# B&R Automation Studio project RTFProj
Automation Studio 4.2.10.53 SP; technology packages: mapp 1.60.1, mappView 1.3.1, TextSystem 

## Configuration RTFProjRG

CPU 5PPC2100.BY44-000, AutomationRuntime B4.26, Build 4.1.2, Vc not used, Safety 1.10

### Task classes (Cpu.sw)
```
Cyclic#1 (cycle 2000 us, tolerance 0 us):
  table_foot <- Real_Game.Technology.table_football.prg
Cyclic#4 (cycle 100000 us, tolerance 100000 us):
  Client <- Connection.Client.prg
DataObjects: assl1, Arnc0sys, Acp10sys
NcDataObjects: acp10etxen <- ACP10_ETXEN.acp10etxen.dob, rotaryFWa <- Real_Game.Motion.rotaryFWobj.rotaryFWa.dob, rotaryFWi <- Real_Game.Motion.rotaryFWobj.rotaryFWi.dob, rotaryMDa <- Real_Game.Motion.rotaryMDobj.rotaryMDa.dob, rotaryMDi <- Real_Game.Motion.rotaryMDobj.rotaryMDi.dob, linearFWa <- Real_Game.Motion.linearFWobj.linearFWa.dob, linearFWi <- Real_Game.Motion.linearFWobj.linearFWi.dob, linearMDa <- Real_Game.Motion.linearMDobj.linearMDa.dob, linearMDi <- Real_Game.Motion.linearMDobj.linearMDi.dob, rotDFa <- Real_Game.Motion.rotDFobj.rotDFa.dob, rotDFi <- Real_Game.Motion.rotDFobj.rotDFi.dob, rotDFVa <- Real_Game.Motion.rotDFVobj.rotDFVa.dob, rotDFVi <- Real_Game.Motion.rotDFVobj.rotDFVi.dob, rotGKa <- Real_Game.Motion.rotGKobj.rotGKa.dob, rotGKi <- Real_Game.Motion.rotGKobj.rotGKi.dob, linDFa <- Real_Game.Motion.linDFobj.linDFa.dob, linDFi <- Real_Game.Motion.linDFobj.linDFi.dob, linDFVa <- Real_Game.Motion.linDFVobj.linDFVa.dob, linDFVi <- Real_Game.Motion.linDFVobj.linDFVi.dob, linGKa <- Real_Game.Motion.linGKobj.linGKa.dob, linGKi <- Real_Game.Motion.linGKobj.linGKi.dob
Binaries: arsvcreg, mvLoader, TCData, udbdef, Linear, iomap, OpcUaMap, sysconf, Config, TC, Config_1, ashwd, asfw, User, arconfig, Role, Rotary, Acp10map, acp10cfg, Arnc0map, arnc0cfg
Libraries: operator, runtime, AsIecCon, sys_lib, astime, AsArSdm, AsWStr, asstring, DataObj, AsArLog, FileIO, AsArProf, AsMem, brsystem, standard, rp_funcx1, GoalKeeper, AsBrStr, IecCheck, MTTypes, MpCom, MpAlarmX, MTBasics, AsSafety, AsXml, MpAxis, Acp10_MC, Acp10man, NcGlobal, Acp10par, RO_Sensors, Camera, Bar_Light, AsUDP, powerlnk, areventlog
```

### Hardware
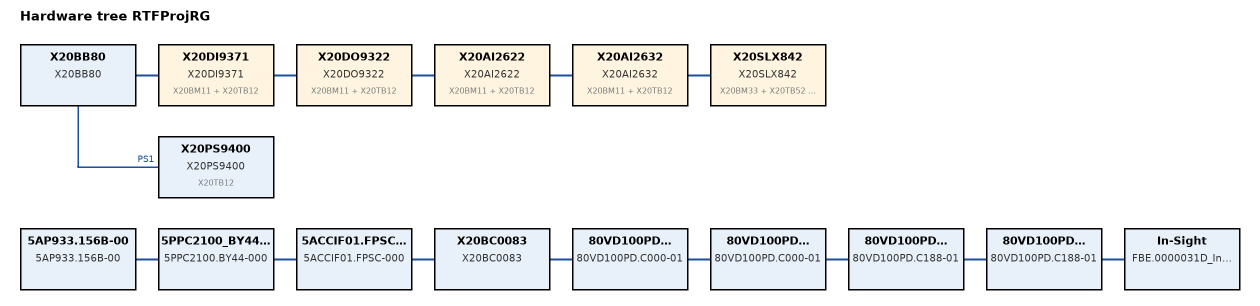
```
5ACCIF01.FPSC-000 : 5ACCIF01.FPSC-000 v1.2.1.0  [SL -> 5PPC2100_BY44_000.SL1]
  Connector IF1:
    Channel1
    ChannelID1 = ACP10_MC_BROADCAST
    ChannelType1 = OCTET[96]
5AP933.156B-00 : 5AP933.156B-00 v1.4.0.1
5PPC2100_BY44_000 : 5PPC2100.BY44-000 v1.2.4.0  [SY -> 5AP933.156B-00.SY1]
  Connector IF3:
    ActivateDevice = 1
  AutomationRuntime = AR010
  ConfigurationID = RTFProj_Config1
  TimerDeviceType = EPLX2X
  TimerDevice = 5ACCIF01.FPSC-000.IF1
  TaskClassIdleTime = 2000
  Cyclic1Duration = 2000
  Cyclic1Tolerance = 0
  Cyclic2Duration = 10000
  Cyclic2Tolerance = 10000
  Cyclic3Duration = 50000
  Cyclic3Tolerance = 50000
  Cyclic4Duration = 100000
  Cyclic4Tolerance = 100000
  Cyclic5Duration = 200000
  Cyclic5Tolerance = 200000
  Cyclic6Duration = 500000
  Cyclic6Tolerance = 500000
  Cyclic7Duration = 1000000
  Cyclic7Tolerance = 1000000
  Cyclic8Duration = 10000
  Cyclic8Tolerance = 30000000
  ActivateOpcUa = 1
  OpcUa_Security_SoftwareCertificates = 
80VD100PD.C000-01 : 80VD100PD.C000-01 v2.0.1.0  [PLK1 -> X20BC0083.PLK2 (NodeNumber=2); PLK2 -> 80VD100PD.C000-01a.PLK1 (NodeNumber=2)]
  BothEndSwitchesAreNormallyOpen_r1 = on
  QuickStopIsNormallyOpen_r1 = on
  BothEndSwitchesAreNormallyOpen_r2 = on
  QuickStopIsNormallyOpen_r2 = on
80VD100PD.C000-01a : 80VD100PD.C000-01 v2.0.1.0  [PLK1 -> 80VD100PD.C000-01.PLK2 (NodeNumber=4); PLK2 -> 80VD100PD.C188-01.PLK1 (NodeNumber=4)]
  BothEndSwitchesAreNormallyOpen_r1 = on
  QuickStopIsNormallyOpen_r1 = on
  BothEndSwitchesAreNormallyOpen_r2 = on
  QuickStopIsNormallyOpen_r2 = on
80VD100PD.C188-01 : 80VD100PD.C188-01 v2.0.1.0  [PLK1 -> 80VD100PD.C000-01a.PLK2 (NodeNumber=3); PLK2 -> 80VD100PD.C188-01a.PLK1 (NodeNumber=3)]
  BothEndSwitchesAreNormallyOpen_r1 = on
  QuickStopIsNormallyOpen_r1 = on
  BothEndSwitchesAreNormallyOpen_r2 = on
  QuickStopIsNormallyOpen_r2 = on
80VD100PD.C188-01a : 80VD100PD.C188-01 v2.0.1.0  [PLK1 -> 80VD100PD.C188-01.PLK2 (NodeNumber=5); PLK2 -> In-Sight.PLK1 (NodeNumber=5)]
  BothEndSwitchesAreNormallyOpen_r1 = on
  QuickStopIsNormallyOpen_r1 = on
  BothEndSwitchesAreNormallyOpen_r2 = on
  QuickStopIsNormallyOpen_r2 = on
In-Sight : FBE.0000031D_In-Sight-7000 v4.8.0 (OrderNumber=In-Sight)  [PLK1 -> 80VD100PD.C188-01a.PLK2 (NodeNumber=6)]
  Supervision = off
  p2000s01_direction = wo
  p2000s02_direction = wo
  p2001s01_direction = ro
  p2001s02_direction = ro
  p2001s03_direction = ro
  p2010s02_direction = ro
  p2011s01_direction = ro
  p2011s02_direction = ro
  p2011s03_direction = ro
  p2011s04_direction = ro
  p2021s01_direction = wo
X20AI2622 : X20AI2622 v1.0.3.1  [SS1 -> X20TB12c.SS; SL -> X20BM11b.SL1]
  Supervision = off
  ChannelType01 = 4 to 20mA
  ChannelType02 = 4 to 20mA
X20AI2632 : X20AI2632 v1.1.5.1  [SS1 -> X20TB12d.SS; SL -> X20BM11c.SL1]
  ChannelType01 = 0 to 20mA
  ChannelType02 = 0 to 20mA
X20BB80 : X20BB80 v1.0.0.2
X20BC0083 : X20BC0083 v2.5.2.0  [PLK1 -> 5ACCIF01.FPSC-000.IF1 (NodeNumber=1); PLK2 -> 80VD100PD.C000-01.PLK1 (NodeNumber=1); SL -> X20BB80.SL1]
  Supervision = off
X20BM11 : X20BM11 v1.0.0.1  [X2X1 -> X20BB80.IF1]
X20BM11a : X20BM11 v1.0.0.1  [X2X1 -> X20BM11.X2X2]
X20BM11b : X20BM11 v1.0.0.1  [X2X1 -> X20BM11a.X2X2]
X20BM11c : X20BM11 v1.0.0.1  [X2X1 -> X20BM11b.X2X2]
X20BM33 : X20BM33 v1.0.0.4  [X2X1 -> X20BM11c.X2X2]
X20DI9371 : X20DI9371 v1.0.1.3  [SS1 -> X20TB12a.SS; SL -> X20BM11.SL1]
  Supervision = off
X20DO9322 : X20DO9322 v1.0.3.0  [SS1 -> X20TB12b.SS; SL -> X20BM11a.SL1]
  Supervision = off
X20PS9400 : X20PS9400 v1.0.2.4  [SS1 -> X20TB12.SS; PS -> X20BB80.PS1]
  Supervision = off
X20SLX842 : X20SLX842 v1.10.3.1  [SS1 -> X20TB52.SS; SS2 -> X20TB52a.SS; SL -> X20BM33.SL1]
  SafeProject = SafeLOGIC-1
  SafeDesigner = 4.2.2.18
  DigitalOutput01 = viaSafeLOGIC
  DigitalOutput02 = viaSafeLOGIC
  DigitalOutput03 = viaSafeLOGIC
  DigitalOutput04 = viaSafeLOGIC
X20TB12 : X20TB12 v1.0.0.0
X20TB12a : X20TB12 v1.0.0.0
X20TB12b : X20TB12 v1.0.0.0
X20TB12c : X20TB12 v1.0.0.0
X20TB12d : X20TB12 v1.0.0.0
X20TB52 : X20TB52 v1.0.0.1
X20TB52a : X20TB52 v1.0.0.1
```

### IoMap.iom - 5PPC2100_BY44_000/IoMap.iom
```iecst
VAR_CONFIG
	::cam_det.InSight.ModuleOk AT %IX."In-Sight".ModuleOk;
	::cam_det.InSight.Control_I2000_S01 AT %QD."In-Sight".Control_I2000_S01;
	::cam_det.InSight.Status_I2001_S01 AT %ID."In-Sight".Status_I2001_S01;
	::cam_det.InSight.InspectionResults_I2011_S01 AT %ID."In-Sight".InspectionResults_I2011_S01; (*X*)
	::cam_det.InSight.InspectionResults_I2011_S02 AT %ID."In-Sight".InspectionResults_I2011_S02; (*Y*)
	::GoalKeeper_0.DI9371.DigitalInput_1 AT %IX."X20DI9371".DigitalInput05;
	::GoalKeeper_0.DI9371.ModuleOk AT %IX."X20DI9371".ModuleOk;
	::Light_0.DO9322.ModuleOK AT %IX."X20DO9322".ModuleOk;
	::Light_0.DO9322.DigitalOutput AT %QX."X20DO9322".DigitalOutput01;
	::GoalKeeper_0.DI9371.DigitalInput_2 AT %IX."X20DI9371".DigitalInput06;
	Cyclic#1.::table_foot:reset_safetyESTOP AT %QX."X20SLX842".BOOL101;
	Cyclic#1.::table_foot:ESTOP AT %IX."X20SLX842".SafeDigitalInput03;
	Cyclic#1.::table_foot:OSSD2 AT %IX."X20SLX842".SafeDigitalInput02;
	Cyclic#1.::table_foot:SAFETY_MODUL_OK AT %IX."X20SLX842".ModuleOk;
	::table_foot:dpA.ActPosSens[0] AT %IW."X20AI2632".AnalogInput01;
	::table_foot:dpA.ActPosSens[1] AT %IW."X20AI2632".AnalogInput02;
	::table_foot:dpA.ActPosSens[3] AT %IW."X20AI2622".AnalogInput01;
	::table_foot:dpA.ActPosSens[2] AT %IW."X20AI2622".AnalogInput02;
	::cam_det.InSight.InspectionResults_I2011_S03 AT %ID."In-Sight".InspectionResults_I2011_S03;
	::cam_det.InSight.InspectionResults_I2011_S04 AT %ID."In-Sight".InspectionResults_I2011_S04;
	::cam_det.InSight.UserData_I2021_S01 AT %QD."In-Sight".UserData_I2021_S01;
	::table_foot:dpA.ReflexSensStatus[3] AT %IX."X20DI9371".DigitalInput01;
	::table_foot:dpA.ReflexSensStatus[2] AT %IX."X20DI9371".DigitalInput02;
	::table_foot:dpA.ReflexSensStatus[0] AT %IX."X20DI9371".DigitalInput03;
	::table_foot:dpA.ReflexSensStatus[1] AT %IX."X20DI9371".DigitalInput04;
END_VAR
```

### Acp10cfg.ncc - 5PPC2100_BY44_000/Motion/Acp10cfg.ncc
```
NcConfiguration (Version=3.16.2, NcSwId=Acp10)
  ACP10CF1_typ:
    cnt_nettrc_rec_drive = 1500
    bufsize_trace_upload = 1200
    tc_nc_man_task = Cyclic #1
    glob_pv_as_ncobject = Yes
    ncsys_dl_broadcast = Yes
    ncsys_dl_acp_reset = Yes
    safemc_log_err_to_ax = Yes
    network_init:
      ncsw_init_execute = Yes
      automatic_execute = Yes
      node_nr_warning = Yes
      net_err_before_ncact = Yes
    nettrc:
      enter_parsecrec = Yes
      enter_ncaction = Yes
      save_ring_startidx = Yes
    cam_prof_download:
      cam_dat_dl_parallel = No
      tc_cam_dl_parallel = Task class for NC Manager task
    plk_if[0]:
      if_name = SL1.IF1
      tc_CycDat_PLCopen = Task class for NC Manager task
      mc_broadcast_extdat = No
```

### Acp10map.ncm - 5PPC2100_BY44_000/Motion/Acp10map.ncm
```
NcMapping (NcSwId=Acp10, DisabledNodesAreHidden=False)
  NcObject 80VD100PD.C000-01a_ncV_AXIS1 (ModuleId=80VD100PD.C000-01a, Type=ncV_AXIS, Channel=1, Disabled=TRUE, ModuleDisabled=FALSE)
  NcObject 80VD100PD.C000-01a_ncV_AXIS2 (ModuleId=80VD100PD.C000-01a, Type=ncV_AXIS, Channel=2, Disabled=TRUE, ModuleDisabled=FALSE)
  NcObject 80VD100PD.C188-01a_ncV_AXIS1 (ModuleId=80VD100PD.C188-01a, Type=ncV_AXIS, Channel=1, Disabled=TRUE, ModuleDisabled=FALSE)
  NcObject 80VD100PD.C188-01a_ncV_AXIS2 (ModuleId=80VD100PD.C188-01a, Type=ncV_AXIS, Channel=2, Disabled=TRUE, ModuleDisabled=FALSE)
  NcObject linearFW (ModuleId=80VD100PD.C188-01a, Type=ncAXIS, Channel=2, AcoposSimulation=Off, InitParameter=linearFWi, AcoposParameter=linearFWa, Disabled=FALSE, ModuleDisabled=FALSE)
  NcObject linearMD (ModuleId=80VD100PD.C188-01a, Type=ncAXIS, Channel=1, AcoposSimulation=Off, InitParameter=linearMDi, AcoposParameter=linearMDa, Disabled=FALSE, ModuleDisabled=FALSE)
  NcObject rotaryFW (ModuleId=80VD100PD.C000-01a, Type=ncAXIS, Channel=2, AcoposSimulation=Off, InitParameter=rotaryFWi, AcoposParameter=rotaryFWa, Disabled=FALSE, ModuleDisabled=FALSE)
  NcObject rotaryMD (ModuleId=80VD100PD.C000-01a, Type=ncAXIS, Channel=1, AcoposSimulation=Off, InitParameter=rotaryMDi, AcoposParameter=rotaryMDa, Disabled=FALSE, ModuleDisabled=FALSE)
  NcObject rotGK (ModuleId=80VD100PD.C000-01, Type=ncAXIS, Channel=1, AcoposSimulation=Off, InitParameter=rotGKi, AcoposParameter=rotGKa, Disabled=FALSE, ModuleDisabled=FALSE)
  NcObject rotDF (ModuleId=80VD100PD.C000-01, Type=ncAXIS, Channel=2, AcoposSimulation=Off, InitParameter=rotDFi, AcoposParameter=rotDFa, Disabled=FALSE, ModuleDisabled=FALSE)
  NcObject 80VD100PD.C000-01_ncV_AXIS1 (ModuleId=80VD100PD.C000-01, Type=ncV_AXIS, Channel=1, Disabled=TRUE, ModuleDisabled=FALSE)
  NcObject rotDFV (ModuleId=80VD100PD.C000-01, Type=ncV_AXIS, Channel=2, InitParameter=rotDFVi, AcoposParameter=rotDFVa, Disabled=FALSE, ModuleDisabled=FALSE)
  NcObject linGK (ModuleId=80VD100PD.C188-01, Type=ncAXIS, Channel=1, AcoposSimulation=Off, InitParameter=linGKi, AcoposParameter=linGKa, Disabled=FALSE, ModuleDisabled=FALSE)
  NcObject linDF (ModuleId=80VD100PD.C188-01, Type=ncAXIS, Channel=2, AcoposSimulation=Off, InitParameter=linDFi, AcoposParameter=linDFa, Disabled=FALSE, ModuleDisabled=FALSE)
  NcObject 80VD100PD.C188-01_ncV_AXIS1 (ModuleId=80VD100PD.C188-01, Type=ncV_AXIS, Channel=1, Disabled=TRUE, ModuleDisabled=FALSE)
  NcObject linDFV (ModuleId=80VD100PD.C188-01, Type=ncV_AXIS, Channel=2, InitParameter=linDFVi, AcoposParameter=linDFVa, Disabled=FALSE, ModuleDisabled=FALSE)
```

- Safety project (password-protected, skipped)

### Config.mpalarmxcore - 5PPC2100_BY44_000/mapp/MpAlaramX/Config.mpalarmxcore
```
Element gAlarmXCoreR (Type=mpalarmxcore)
```

### Config_1.mpalarmxhistory - 5PPC2100_BY44_000/mapp/MpAlaramX/Config_1.mpalarmxhistory
```
Element gAlarmXHistoryR (Type=mpalarmxhistory)
```

### Linear.mpaxisbasic - 5PPC2100_BY44_000/mapp/MpAxisBasic/Linear.mpaxisbasic
```
Element gk_mappAxisLR (Type=mpaxisbasic)
Element df_mappAxisLR (Type=mpaxisbasic)
Element md_mappAxisLR (Type=mpaxisbasic)
Element fw_mappAxisLR (Type=mpaxisbasic)
```

### Rotary.mpaxisbasic - 5PPC2100_BY44_000/mapp/MpAxisBasic/Rotary.mpaxisbasic
```
Element gk_mappAxisRR (Type=mpaxisbasic)
Element df_mappAxisRR (Type=mpaxisbasic)
Element md_mappAxisRR (Type=mpaxisbasic)
Element fw_mappAxisRR (Type=mpaxisbasic)
```

## Configuration Simulation

CPU , AutomationRuntime B4.26, Build 4.1.2, Safety 1.10

### Task classes (Cpu.sw)
```
Cyclic#1 (cycle 2000 us, tolerance 0 us):
  simulation <- Simulation.Technology.simulation.prg
  sim_cam_se <- Simulation.Technology.sim_cam_sens_sd_s.prg [disabled]
DataObjects: Acp10sys, Arnc0sys
NcDataObjects: dfRotSa <- Simulation.Motion.dfRotSobj.dfRotSa.dob, dfRotSi <- Simulation.Motion.dfRotSobj.dfRotSi.dob, gkRotSa <- Simulation.Motion.gkRotSobj.gkRotSa.dob, gkRotSi <- Simulation.Motion.gkRotSobj.gkRotSi.dob, dfLinSa <- Simulation.Motion.dfLinSobj.dfLinSa.dob, dfLinSi <- Simulation.Motion.dfLinSobj.dfLinSi.dob, gkLinSa <- Simulation.Motion.gkLinSobj.gkLinSa.dob, gkLinSi <- Simulation.Motion.gkLinSobj.gkLinSi.dob, fwRotSa <- Simulation.Motion.fwRotSobj.fwRotSa.dob, fwRotSi <- Simulation.Motion.fwRotSobj.fwRotSi.dob, mdRotSa <- Simulation.Motion.mdRotSobj.mdRotSa.dob, mdRotSi <- Simulation.Motion.mdRotSobj.mdRotSi.dob, fwLinSa <- Simulation.Motion.fwLinSobj.fwLinSa.dob, fwLinSi <- Simulation.Motion.fwLinSobj.fwLinSi.dob, mdLinSa <- Simulation.Motion.mdLinSobj.mdLinSa.dob, mdLinSi <- Simulation.Motion.mdLinSobj.mdLinSi.dob
Binaries: arsvcreg, mvLoader, TCData, udbdef, Linear, iomap, sysconf, Config, Config_1, ashwd, asfw, User, arconfig, Role, Rotary, Acp10map, acp10cfg, Core, History
Libraries: AsIecCon, astime, MpCom, MpAlarmX, Runtime, AsArSdm, rp_funcx1, AsWStr, asstring, Acp10man, Acp10par, NcGlobal, DataObj, AsArLog, sys_lib, FileIO, AsArProf, AsMem, brsystem, Acp10_MC, AsBrStr, IecCheck, AsSafety, AsXml, standard, MTBasics, MTTypes, MpAxis, powerlnk, areventlog, Acp10sim
```

### Hardware
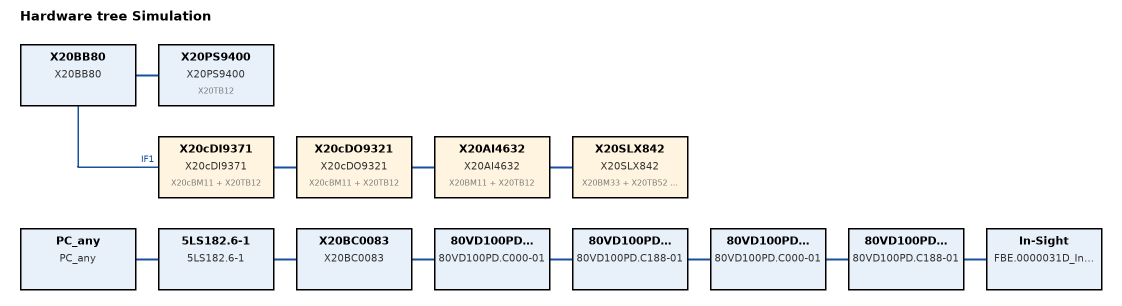
```
5LS182.6-1 : 5LS182.6-1 v1.3.0.0  [SL -> PC_any.SL1]
  Connector IF1:
    EplInterfaceRedundant = 0
    EplEthInterfaceRedundant = 0
80VD100PD.C000-01 : 80VD100PD.C000-01 v2.0.1.0  [PLK1 -> X20BC0083.PLK2 (NodeNumber=2); PLK2 -> 80VD100PD.C188-01.PLK1 (NodeNumber=2)]
  BothEndSwitchesAreNormallyOpen_r1 = on
  QuickStopIsNormallyOpen_r1 = on
  BothEndSwitchesAreNormallyOpen_r2 = on
  QuickStopIsNormallyOpen_r2 = on
80VD100PD.C000-01a : 80VD100PD.C000-01 v2.0.1.0  [PLK1 -> 80VD100PD.C188-01.PLK2 (NodeNumber=4); PLK2 -> 80VD100PD.C188-01a.PLK1 (NodeNumber=4)]
  BothEndSwitchesAreNormallyOpen_r1 = on
  QuickStopIsNormallyOpen_r1 = on
  BothEndSwitchesAreNormallyOpen_r2 = on
  QuickStopIsNormallyOpen_r2 = on
80VD100PD.C188-01 : 80VD100PD.C188-01 v2.0.1.0  [PLK1 -> 80VD100PD.C000-01.PLK2 (NodeNumber=3); PLK2 -> 80VD100PD.C000-01a.PLK1 (NodeNumber=3)]
  BothEndSwitchesAreNormallyOpen_r1 = on
  QuickStopIsNormallyOpen_r1 = on
  BothEndSwitchesAreNormallyOpen_r2 = on
  QuickStopIsNormallyOpen_r2 = on
80VD100PD.C188-01a : 80VD100PD.C188-01 v2.0.1.0  [PLK1 -> 80VD100PD.C000-01a.PLK2 (NodeNumber=5); PLK2 -> In-Sight.PLK1 (NodeNumber=5)]
  BothEndSwitchesAreNormallyOpen_r1 = on
  QuickStopIsNormallyOpen_r1 = on
  BothEndSwitchesAreNormallyOpen_r2 = on
  QuickStopIsNormallyOpen_r2 = on
In-Sight : FBE.0000031D_In-Sight-7000 v4.8.0 (Disabled=true, OrderNumber=In-Sight)  [PLK1 -> 80VD100PD.C188-01a.PLK2 (NodeNumber=6)]
  p2000s01_direction = wo
  p2000s02_direction = wo
  p2001s01_direction = ro
  p2001s02_direction = ro
  p2001s03_direction = ro
  p2010s02_direction = ro
  p2011s01_direction = ro
  p2011s02_direction = ro
PC_any : PC_any v1.1.0.0 (OrderNumber=PC)
  ConfigurationID = rp_masterThesis_SoccerTable_Simulation
  SystemTick = 2000
  Cyclic1Duration = 2000
  Cyclic1Tolerance = 0
  Cyclic2Duration = 200000
  Cyclic2Tolerance = 10000000
  Cyclic3Duration = 500000
  Cyclic3Tolerance = 10000000
  Cyclic4Duration = 1000000
  Cyclic4Tolerance = 10000000
  Cyclic5Duration = 2000000
  Cyclic5Tolerance = 10000000
  Cyclic6Duration = 3000000
  Cyclic6Tolerance = 12000000
  Cyclic7Duration = 4000000
  Cyclic7Tolerance = 12000000
  Cyclic8Duration = 5000000
  Cyclic8Tolerance = 30000000
  FileDevice1
  FileDeviceName1 = EXPORT_HISTORY
  FileDevicePath1 = C:\Temp\AlarmX\SOCCER_TABLE
  ActivateOpcUa = 1
  OpcUa_Security_SoftwareCertificates = 
  Temp.ProjectDirectory = C:\projects\ProjectRealST\
  Temp.ConfigurationName = Simulation
X20AI4632 : X20AI4632 v1.1.3.1  [SS1 -> X20TB12c.SS; SL -> X20BM11.SL1]
X20BB80 : X20BB80 v1.0.0.2
X20BC0083 : X20BC0083 v2.5.2.0  [PLK1 -> 5LS182.6-1.IF1 (NodeNumber=1); PLK2 -> 80VD100PD.C000-01.PLK1 (NodeNumber=1); SL -> X20BB80.SL1]
X20BM11 : X20BM11 v1.0.0.1  [X2X1 -> X20cBM11a.X2X2]
X20BM33 : X20BM33 v1.0.0.4  [X2X1 -> X20BM11.X2X2]
X20PS9400 : X20PS9400 v1.0.2.4  [SS1 -> X20TB12.SS; PS -> X20BB80.PS1]
X20SLX842 : X20SLX842 v1.10.1.2  [SS1 -> X20TB52.SS; SS2 -> X20TB52a.SS; SL -> X20BM33.SL1]
  SafeProject = SafeLOGIC-1
  SafeDesigner = 4.2.2.18
X20TB12 : X20TB12 v1.0.0.0
X20TB12a : X20TB12 v1.0.0.0
X20TB12b : X20TB12 v1.0.0.0
X20TB12c : X20TB12 v1.0.0.0
X20TB52 : X20TB52 v1.0.0.1
X20TB52a : X20TB52 v1.0.0.1
X20cBM11 : X20cBM11 v1.0.0.0  [X2X1 -> X20BB80.IF1]
X20cBM11a : X20cBM11 v1.0.0.0  [X2X1 -> X20cBM11.X2X2]
X20cDI9371 : X20cDI9371 v1.0.0.1  [SS1 -> X20TB12a.SS; SL -> X20cBM11.SL1]
X20cDO9321 : X20cDO9321 v1.0.2.0  [SS1 -> X20TB12b.SS; SL -> X20cBM11a.SL1]
```

### Acp10cfg.ncc - PC_any/Motion/Acp10cfg.ncc
```
NcConfiguration (Version=3.13.0, NcSwId=Acp10)
  ACP10CF1_typ:
    cnt_nettrc_rec_drive = 1500
    bufsize_trace_upload = 1200
    tc_nc_man_task = Cyclic #1
    glob_pv_as_ncobject = Yes
    ncsys_dl_broadcast = Yes
    ncsys_dl_acp_reset = Yes
    safemc_log_err_to_ax = Yes
    network_init:
      ncsw_init_execute = Yes
      automatic_execute = No
      node_nr_warning = Yes
      net_err_before_ncact = Yes
    nettrc:
      enter_parsecrec = Yes
      enter_ncaction = Yes
      save_ring_startidx = Yes
    cam_prof_download:
      cam_dat_dl_parallel = No
      tc_cam_dl_parallel = Task class for NC Manager task
    plk_if[0]:
      if_name = SL1.IF1
      tc_CycDat_PLCopen = Task class for NC Manager task
      mc_broadcast_extdat = No
```

### Acp10map.ncm - PC_any/Motion/Acp10map.ncm
```
NcMapping (NcSwId=Acp10, DisabledNodesAreHidden=False)
  NcObject gkRotS (ModuleId=80VD100PD.C000-01, Type=ncAXIS, Channel=1, AcoposSimulation=Off, InitParameter=gkRotSi, AcoposParameter=gkRotSa, Disabled=FALSE, ModuleDisabled=FALSE)
  NcObject dfRotS (ModuleId=80VD100PD.C000-01, Type=ncAXIS, Channel=2, AcoposSimulation=Off, InitParameter=dfRotSi, AcoposParameter=dfRotSa, Disabled=FALSE, ModuleDisabled=FALSE)
  NcObject 80VD100PD.C000-01_ncV_AXIS1 (ModuleId=80VD100PD.C000-01, Type=ncV_AXIS, Channel=1, Disabled=TRUE, ModuleDisabled=FALSE)
  NcObject 80VD100PD.C000-01_ncV_AXIS2 (ModuleId=80VD100PD.C000-01, Type=ncV_AXIS, Channel=2, Disabled=TRUE, ModuleDisabled=FALSE)
  NcObject gkLinS (ModuleId=80VD100PD.C188-01, Type=ncAXIS, Channel=1, AcoposSimulation=Off, InitParameter=gkLinSi, AcoposParameter=gkLinSa, Disabled=FALSE, ModuleDisabled=FALSE)
  NcObject dfLinS (ModuleId=80VD100PD.C188-01, Type=ncAXIS, Channel=2, AcoposSimulation=Off, InitParameter=dfLinSi, AcoposParameter=dfLinSa, Disabled=FALSE, ModuleDisabled=FALSE)
  NcObject 80VD100PD.C188-01_ncV_AXIS1 (ModuleId=80VD100PD.C188-01, Type=ncV_AXIS, Channel=1, Disabled=TRUE, ModuleDisabled=FALSE)
  NcObject 80VD100PD.C188-01_ncV_AXIS2 (ModuleId=80VD100PD.C188-01, Type=ncV_AXIS, Channel=2, Disabled=TRUE, ModuleDisabled=FALSE)
  NcObject mdRotS (ModuleId=80VD100PD.C000-01a, Type=ncAXIS, Channel=1, AcoposSimulation=Off, InitParameter=mdRotSi, AcoposParameter=mdRotSa, Disabled=FALSE, ModuleDisabled=FALSE)
  NcObject fwRotS (ModuleId=80VD100PD.C000-01a, Type=ncAXIS, Channel=2, AcoposSimulation=Off, InitParameter=fwRotSi, AcoposParameter=fwRotSa, Disabled=FALSE, ModuleDisabled=FALSE)
  NcObject 80VD100PD.C000-01a_ncV_AXIS1 (ModuleId=80VD100PD.C000-01a, Type=ncV_AXIS, Channel=1, Disabled=TRUE, ModuleDisabled=FALSE)
  NcObject 80VD100PD.C000-01a_ncV_AXIS2 (ModuleId=80VD100PD.C000-01a, Type=ncV_AXIS, Channel=2, Disabled=TRUE, ModuleDisabled=FALSE)
  NcObject mdLinS (ModuleId=80VD100PD.C188-01a, Type=ncAXIS, Channel=1, AcoposSimulation=Off, InitParameter=mdLinSi, AcoposParameter=mdLinSa, Disabled=FALSE, ModuleDisabled=FALSE)
  NcObject fwLinS (ModuleId=80VD100PD.C188-01a, Type=ncAXIS, Channel=2, AcoposSimulation=Off, InitParameter=fwLinSi, AcoposParameter=fwLinSa, Disabled=FALSE, ModuleDisabled=FALSE)
  NcObject 80VD100PD.C188-01a_ncV_AXIS1 (ModuleId=80VD100PD.C188-01a, Type=ncV_AXIS, Channel=1, Disabled=TRUE, ModuleDisabled=FALSE)
  NcObject 80VD100PD.C188-01a_ncV_AXIS2 (ModuleId=80VD100PD.C188-01a, Type=ncV_AXIS, Channel=2, Disabled=TRUE, ModuleDisabled=FALSE)
```

### Arnc0cfg.ncc - PC_any/Motion/Arnc0cfg.ncc
```
NcConfiguration (Version=3.13.1, NcSwId=Arnc0)
  ARNC0CFG_typ:
    sampling_rate = 4000
    cnt_nettrc_rec_drive = 150
    bufsize_sys_trace = 16#00005000
    enable_mp_log = Yes
    tc_nc_man_task = Cyclic #1
    bg_load = 1
    glob_pv_as_ncobject = Yes
```

### Arnc0map.ncm - PC_any/Motion/Arnc0map.ncm
```
NcMapping (NcSwId=Arnc0)
  NcObject CNC1 (Type=ncCNCSYS, Channel=1, AcoposSimulation=Off, Disabled=TRUE, ModuleDisabled=FALSE)
  NcObject CNC2 (Type=ncCNCSYS, Channel=2, AcoposSimulation=Off, Disabled=TRUE, ModuleDisabled=FALSE)
  NcObject CNC3 (Type=ncCNCSYS, Channel=3, AcoposSimulation=Off, Disabled=TRUE, ModuleDisabled=FALSE)
  NcObject CNC4 (Type=ncCNCSYS, Channel=4, AcoposSimulation=Off, Disabled=TRUE, ModuleDisabled=FALSE)
  NcObject CNC5 (Type=ncCNCSYS, Channel=5, AcoposSimulation=Off, Disabled=TRUE, ModuleDisabled=FALSE)
  NcObject CNC6 (Type=ncCNCSYS, Channel=6, AcoposSimulation=Off, Disabled=TRUE, ModuleDisabled=FALSE)
  NcObject CNC7 (Type=ncCNCSYS, Channel=7, AcoposSimulation=Off, Disabled=TRUE, ModuleDisabled=FALSE)
  NcObject CNC8 (Type=ncCNCSYS, Channel=8, AcoposSimulation=Off, Disabled=TRUE, ModuleDisabled=FALSE)
  NcObject CNC9 (Type=ncCNCSYS, Channel=9, AcoposSimulation=Off, Disabled=TRUE, ModuleDisabled=FALSE)
  NcObject CNC10 (Type=ncCNCSYS, Channel=10, AcoposSimulation=Off, Disabled=TRUE, ModuleDisabled=FALSE)
  NcObject CNC11 (Type=ncCNCSYS, Channel=11, AcoposSimulation=Off, Disabled=TRUE, ModuleDisabled=FALSE)
  NcObject CNC12 (Type=ncCNCSYS, Channel=12, AcoposSimulation=Off, Disabled=TRUE, ModuleDisabled=FALSE)
  NcObject CNC13 (Type=ncCNCSYS, Channel=13, AcoposSimulation=Off, Disabled=TRUE, ModuleDisabled=FALSE)
  NcObject CNC14 (Type=ncCNCSYS, Channel=14, AcoposSimulation=Off, Disabled=TRUE, ModuleDisabled=FALSE)
  NcObject CNC15 (Type=ncCNCSYS, Channel=15, AcoposSimulation=Off, Disabled=TRUE, ModuleDisabled=FALSE)
  NcObject CNC16 (Type=ncCNCSYS, Channel=16, AcoposSimulation=Off, Disabled=TRUE, ModuleDisabled=FALSE)
  NcObject CNC17 (Type=ncCNCSYS, Channel=17, AcoposSimulation=Off, Disabled=TRUE, ModuleDisabled=FALSE)
  NcObject CNC18 (Type=ncCNCSYS, Channel=18, AcoposSimulation=Off, Disabled=TRUE, ModuleDisabled=FALSE)
  NcObject CNC19 (Type=ncCNCSYS, Channel=19, AcoposSimulation=Off, Disabled=TRUE, ModuleDisabled=FALSE)
  NcObject CNC20 (Type=ncCNCSYS, Channel=20, AcoposSimulation=Off, Disabled=TRUE, ModuleDisabled=FALSE)
  NcObject CNC21 (Type=ncCNCSYS, Channel=21, AcoposSimulation=Off, Disabled=TRUE, ModuleDisabled=FALSE)
  NcObject CNC22 (Type=ncCNCSYS, Channel=22, AcoposSimulation=Off, Disabled=TRUE, ModuleDisabled=FALSE)
  NcObject CNC23 (Type=ncCNCSYS, Channel=23, AcoposSimulation=Off, Disabled=TRUE, ModuleDisabled=FALSE)
  NcObject CNC24 (Type=ncCNCSYS, Channel=24, AcoposSimulation=Off, Disabled=TRUE, ModuleDisabled=FALSE)
```

### Config.mpalarmxcore - PC_any/mapp/MpAlaramX/Config.mpalarmxcore
```
Element gAlarmXCoreS (Type=mpalarmxcore)
```

### Config_1.mpalarmxhistory - PC_any/mapp/MpAlaramX/Config_1.mpalarmxhistory
```
Element gAlarmXHistoryS (Type=mpalarmxhistory)
```

### Linear.mpaxisbasic - PC_any/mapp/MpAxisBasic/Linear.mpaxisbasic
```
Element gk_mappAxisLS (Type=mpaxisbasic)
Element df_mappAxisLS (Type=mpaxisbasic)
Element md_mappAxisLS (Type=mpaxisbasic)
Element fw_mappAxisLS (Type=mpaxisbasic)
```

### Rotary.mpaxisbasic - PC_any/mapp/MpAxisBasic/Rotary.mpaxisbasic
```
Element gk_mappAxisRS (Type=mpaxisbasic)
Element df_mappAxisRS (Type=mpaxisbasic)
Element md_mappAxisRS (Type=mpaxisbasic)
Element fw_mappAxisRS (Type=mpaxisbasic)
```

## Logical view

Binary libraries used (declarations not repeated): operator, runtime, AsIecCon, sys_lib, astime, AsArSdm, AsWStr, asstring, DataObj, AsArLog, FileIO, AsArProf, AsMem, brsystem, standard, AsBrStr, MTTypes 1.03.0, MTBasics 2.21.0, AsSafety, AsXml, Acp10man 3.16.2, Acp10par 3.16.2, NcGlobal 3.16.2, Acp10_MC 3.16.2, MpCom 1.60.1, MpAxis 1.60.1, MpAlarmX 1.60.1, Acp10sim 3.16.2, AsUDP

### Global.var - Global variables
```iecst
VAR
	adress : STRING[20] := '172.25.15.68';
	port : UINT := 11000;
	path : STRING[200] := 'C:\\Program Files (x86)\\Google\\Chrome\\Application\\chrome.exe';
	arguments : STRING[200] := '--start-fullscreen http://172.25.15.67:81/index.html?visuId=RSTSIMPROJ';
END_VAR
```

### Package Logical/Libraries - Global libraries

### Package Logical/Libraries/rp_library - Roman Parák Library

### Library Logical/Libraries/rp_library/rp_funcx1 (ANSIC)
Depends on: MpAlarmX

#### rp_funcx1.fun - Exported functions and function blocks
```iecst
FUNCTION_BLOCK start_virtualAxis
	VAR_INPUT
		Enable : BOOL;
		start_btn : BOOL;
		axis_name : REFERENCE TO MpAxisBasic;
		axis_param : REFERENCE TO MpAxisBasicParType;
	END_VAR
	VAR_OUTPUT
		succesfully : BOOL;
	END_VAR
	VAR
		Internal : internal_startAxisR;
	END_VAR
END_FUNCTION_BLOCK

FUNCTION_BLOCK measurement_ofScore (*TODO: Add your comment here*) (*$GROUP=User,$CAT=User,$GROUPICON=User.png,$CATICON=User.png*)
	VAR_INPUT
		Enable : BOOL;
		start_measurement : BOOL;
		exit_game : BOOL;
		pause : BOOL;
		restart_measurement : BOOL;
		sens_wicket_CPU : BOOL;
		sens_wicket_HUM : BOOL;
		PLAYER1_NAME : STRING[30];
		PLAYER2_NAME : STRING[30];
	END_VAR
	VAR_OUTPUT
		Error : BOOL;
		probability_CPU : USINT;
		probability_HUM : USINT;
		count_goals_CPU : USINT;
		match_informations : match_info;
		team_nameCPU : STRING[30];
		team_nameHUM : STRING[30];
		count_goals_HUM : USINT;
	END_VAR
	VAR
		Internal : internal_machtInfo;
	END_VAR
END_FUNCTION_BLOCK

FUNCTION_BLOCK axes_control (*TODO: Add your comment here*) (*$GROUP=User,$CAT=User,$GROUPICON=User.png,$CATICON=User.png*)
	VAR_INPUT
		Enable : BOOL;
		start_move : BOOL;
		linear_axis_cyclic : REFERENCE TO MpAxisCyclicSet;
		linear_axis_param : REFERENCE TO MpAxisCyclicSetParType;
		linear_param : param_ac;
		rotary_axis_cyclic : REFERENCE TO MpAxisCyclicSet;
		rotary_axis_param : REFERENCE TO MpAxisCyclicSetParType;
		rotary_param : param_ac;
	END_VAR
	VAR_OUTPUT
		successfully : BOOL;
	END_VAR
	VAR
		Internal : internal_controlAxis;
	END_VAR
END_FUNCTION_BLOCK

FUNCTION_BLOCK calculete_min
	VAR_INPUT
		cmp_num : ARRAY[0..4] OF REAL;
	END_VAR
	VAR_OUTPUT
		index : USINT;
		number : REAL;
	END_VAR
END_FUNCTION_BLOCK

FUNCTION_BLOCK choosing_rightDummy
	VAR_INPUT
		index : USINT;
		real_cross : REAL;
		max_dispOfD : ARRAY[0..3] OF REAL;
		min_dispOfD : ARRAY[0..3] OF REAL;
		matrix_posOfCPU : ARRAY[0..3,0..4] OF REAL;
	END_VAR
	VAR_OUTPUT
		actual_displacement : REAL;
	END_VAR
END_FUNCTION_BLOCK

FUNCTION_BLOCK arrival_timeOfBall
	VAR_INPUT
		ball1_x : REAL;
		ball1_y : REAL;
		ball2_x : REAL;
		ball2_y : REAL;
		first_reflection_x : REAL;
		first_reflection_y : REAL;
		act_posOfAxesX : ARRAY[0..3] OF REAL;
		act_posOfAxesY : ARRAY[0..3] OF REAL;
		time_B2B : REAL;
		tilted : BOOL;
		count_axesIntersection : ARRAY[0..1] OF USINT;
	END_VAR
	VAR_OUTPUT
		velocity : REAL;
		time_aI : ARRAY[0..3] OF REAL;
	END_VAR
END_FUNCTION_BLOCK

FUNCTION_BLOCK calculate_directionOfTilt
	VAR_INPUT
		ball1_x : REAL;
		ball1_y : REAL;
		ball2_x : REAL;
		ball2_y : REAL;
	END_VAR
	VAR_OUTPUT
		reflection_x : REAL;
		reflection_y : REAL;
		state_ofDirection : USINT;
		specific_direction : STRING[30];
	END_VAR
END_FUNCTION_BLOCK

FUNCTION_BLOCK calculate_nextDirection
	VAR_INPUT
		first_reflection_x : REAL;
		first_reflection_y : REAL;
		ball2_x : REAL;
		ball2_y : REAL;
		state_ofDirection : USINT;
	END_VAR
	VAR_OUTPUT
		second_reflection_x : REAL;
		second_reflection_y : REAL;
	END_VAR
END_FUNCTION_BLOCK

FUNCTION_BLOCK calculation_crossingBall (*TODO: Add your comment here*) (*$GROUP=User,$CAT=User,$GROUPICON=User.png,$CATICON=User.png*)
	VAR_INPUT
		x_positions : ARRAY[0..3] OF REAL;
		ball1_x : REAL;
		ball1_y : REAL;
		ball2_x : REAL;
		ball2_y : REAL;
		first_reflection_x : REAL;
		first_reflection_y : REAL;
		second_reflection_x : REAL;
		second_reflection_y : REAL;
		time_B2B : REAL;
		tilted : BOOL;
	END_VAR
	VAR_OUTPUT
		count_axesIntersection : ARRAY[0..1] OF USINT;
		act_posOfAxesX : ARRAY[0..3] OF REAL;
		act_posOfAxesY : ARRAY[0..3] OF REAL;
		overall_velocity : REAL;
		time_axisIntersection : ARRAY[0..3] OF REAL;
	END_VAR
END_FUNCTION_BLOCK

FUNCTION_BLOCK calculation_displacementOfAxes (*TODO: Add your comment here*) (*$GROUP=User,$CAT=User,$GROUPICON=User.png,$CATICON=User.png*)
	VAR_INPUT
		tilted : BOOL;
		specific_direction : STRING[30];
		count_axesIntersectionHUM : ARRAY[0..1] OF USINT;
		act_posOfAxesCPU_Y : ARRAY[0..3] OF REAL;
		time_axisIntersection : ARRAY[0..3] OF REAL;
		act_displacementCPU : ARRAY[0..3] OF REAL;
		reversed_HUM : ARRAY[0..3] OF BOOL;
		act_posOfDummiesH : ARRAY[0..10] OF REAL;
		act_posOfAxesHUM_Y : ARRAY[0..3] OF REAL;
		x_posOfBall : ARRAY[0..1] OF REAL;
	END_VAR
	VAR_OUTPUT
		displacement : ARRAY[0..3] OF REAL;
		velocity : ARRAY[0..3] OF REAL;
		acceleration : ARRAY[0..3] OF REAL;
		deceleration : ARRAY[0..3] OF REAL;
	END_VAR
END_FUNCTION_BLOCK

FUNCTION_BLOCK calculation_newCrossing
	VAR_INPUT
		specific_direction : STRING[30];
		iteration : USINT;
		reversed_HUM : BOOL;
		predicted_position : REAL;
		act_posOfAxesCPU_Y : ARRAY[0..3] OF REAL;
		act_posOfAxesHUM_Y : ARRAY[0..3] OF REAL;
		x_posOfBall : ARRAY[0..1] OF REAL;
	END_VAR
	VAR_OUTPUT
		new_cross : ARRAY[0..3] OF REAL;
	END_VAR
END_FUNCTION_BLOCK

FUNCTION_BLOCK calculation_posDummies (*TODO: Add your comment here*) (*$GROUP=User,$CAT=User,$GROUPICON=User.png,$CATICON=User.png*)
	VAR_INPUT
		displacement : ARRAY[0..3] OF REAL;
		max_disp : ARRAY[0..3] OF REAL;
		min_disp : ARRAY[0..3] OF REAL;
	END_VAR
	VAR_OUTPUT
		actual_positionsOfDummies : ARRAY[0..10] OF REAL;
		real_displacement : ARRAY[0..3] OF REAL;
	END_VAR
END_FUNCTION_BLOCK

FUNCTION_BLOCK calculation_realCrossing
	VAR_INPUT
		tilted : BOOL;
		specific_direction : STRING[30];
		count_axesIntersectionHUM : ARRAY[0..1] OF USINT;
		act_posOfAxesCPU_Y : ARRAY[0..3] OF REAL;
		reversed_HUM : ARRAY[0..3] OF BOOL;
		act_posOfDummiesH : ARRAY[0..10] OF REAL;
		act_posOfAxesHUM_Y : ARRAY[0..3] OF REAL;
		x_posOfBall : ARRAY[0..1] OF REAL;
	END_VAR
	VAR_OUTPUT
		real_cross : ARRAY[0..3] OF REAL;
	END_VAR
END_FUNCTION_BLOCK

FUNCTION_BLOCK forecast_direction (*TODO: Add your comment here*) (*$GROUP=User,$CAT=User,$GROUPICON=User.png,$CATICON=User.png*)
	VAR_INPUT
		ball1_x : REAL;
		ball1_y : REAL;
		ball2_x : REAL;
		ball2_y : REAL;
	END_VAR
	VAR_OUTPUT
		tilted : BOOL;
		specific_direction : STRING[30];
		first_reflectionX : REAL;
		first_reflectionY : REAL;
		second_reflectionX : REAL;
		second_reflectionY : REAL;
	END_VAR
END_FUNCTION_BLOCK

FUNCTION random_number : INT (*TODO: Add your comment here*) (*$GROUP=User,$CAT=User,$GROUPICON=User.png,$CATICON=User.png*)
	VAR_INPUT
		min_num : INT;
		max_num : INT;
	END_VAR
END_FUNCTION

FUNCTION_BLOCK start_linearAxis (*TODO: Add your comment here*) (*$GROUP=User,$CAT=User,$GROUPICON=User.png,$CATICON=User.png*)
	VAR_INPUT
		Enable : BOOL;
		start_btn : BOOL;
		axis_name : REFERENCE TO MpAxisBasic;
		axis_param : REFERENCE TO MpAxisBasicParType;
		velocity : REAL;
		max_leftPosition : REAL;
	END_VAR
	VAR_OUTPUT
		succesfully : BOOL;
	END_VAR
	VAR
		Internal : internal_startAxisR;
	END_VAR
END_FUNCTION_BLOCK

FUNCTION_BLOCK start_rotaryAxis (*TODO: Add your comment here*) (*$GROUP=User,$CAT=User,$GROUPICON=User.png,$CATICON=User.png*)
	VAR_INPUT
		Enable : BOOL;
		start_btn : BOOL;
		axis_name : REFERENCE TO MpAxisBasic;
		axis_param : REFERENCE TO MpAxisBasicParType;
		value_ofRotatation : LREAL;
	END_VAR
	VAR_OUTPUT
		succesfully : BOOL;
	END_VAR
	VAR
		Internal : internal_startAxisR;
	END_VAR
END_FUNCTION_BLOCK

FUNCTION_BLOCK err_detection (*TODO: Add your comment here*) (*$GROUP=User,$CAT=User,$GROUPICON=User.png,$CATICON=User.png*)
	VAR_INPUT
		rotary_ERR : ARRAY[0..3] OF BOOL;
		linear_ERR : ARRAY[0..3] OF BOOL;
	END_VAR
	VAR_OUTPUT
		err_detect : BOOL;
	END_VAR
END_FUNCTION_BLOCK

FUNCTION_BLOCK control_temperature (*TODO: Add your comment here*) (*$GROUP=User,$CAT=User,$GROUPICON=User.png,$CATICON=User.png*)
	VAR_INPUT
		temperature_rotary : ARRAY[0..3] OF LREAL;
		temperature_linear : ARRAY[0..3] OF LREAL;
	END_VAR
	VAR_OUTPUT
		high_temp_rotary : ARRAY[0..3] OF BOOL;
		high_temp_linear : ARRAY[0..3] OF BOOL;
		start_cooling_linear : ARRAY[0..3] OF BOOL;
	END_VAR
END_FUNCTION_BLOCK

FUNCTION_BLOCK get_rotationalPostition
	VAR_INPUT
		actual_position : ARRAY[0..3] OF LREAL;
		define_position : ARRAY[0..3] OF LREAL;
	END_VAR
	VAR_OUTPUT
		result : ARRAY[0..3] OF LREAL;
	END_VAR
END_FUNCTION_BLOCK

FUNCTION_BLOCK ball_shooting (*TODO: Add your comment here*) (*$GROUP=User,$CAT=User,$GROUPICON=User.png,$CATICON=User.png*)
	VAR_INPUT
		Enable : BOOL;
		start_shoot : BOOL;
		rotary_axes : REFERENCE TO MpAxisCyclicSet;
	END_VAR
	VAR_OUTPUT
		successfully : BOOL;
	END_VAR
	VAR
		Internal : internal_ballShooting;
	END_VAR
END_FUNCTION_BLOCK

FUNCTION_BLOCK turn_position (*TODO: Add your comment here*) (*$GROUP=User,$CAT=User,$GROUPICON=User.png,$CATICON=User.png*)
	VAR_INPUT
		Enable : BOOL;
		start_turn : BOOL;
		index_ofAxis : USINT;
		linear_axes : REFERENCE TO MpAxisCyclicSet;
		rotary_axes : REFERENCE TO MpAxisCyclicSet;
	END_VAR
	VAR_OUTPUT
		successfully : BOOL;
	END_VAR
	VAR
		Internal : internal_turnPos;
	END_VAR
END_FUNCTION_BLOCK

FUNCTION_BLOCK detect_axisNumber
	VAR_INPUT
		ball1_x : REAL;
		ball2_x : REAL;
	END_VAR
	VAR_OUTPUT
		axis_number : USINT;
	END_VAR
END_FUNCTION_BLOCK

FUNCTION_BLOCK choose_attack_mode
	VAR_INPUT
		axis_number : USINT;
		behind_position : INT;
		before_position : INT;
		ball1_x : REAL;
		ball1_y : REAL;
		ball2_x : REAL;
		ball2_y : REAL;
		actual_positionsOfDummies : ARRAY[0..10] OF REAL;
	END_VAR
	VAR_OUTPUT
		mode : USINT;
	END_VAR
END_FUNCTION_BLOCK

FUNCTION_BLOCK check_attack_mode (*TODO: Add your comment here*) (*$GROUP=User,$CAT=User,$GROUPICON=User.png,$CATICON=User.png*)
	VAR_INPUT
		ball1_x : REAL;
		ball1_y : REAL;
		ball2_x : REAL;
		ball2_y : REAL;
		angle_ofRotation : ARRAY[0..3] OF REAL;
		act_displacement_cpu : ARRAY[0..3] OF REAL;
	END_VAR
	VAR_OUTPUT
		attack_mode : USINT;
		index_ofAxis : USINT;
	END_VAR
END_FUNCTION_BLOCK
```

#### rp_functions.c
```c
/*********************************************************************************************
* B&R Automation - Perfection in Automation (https://www.br-automation.com)
    ******************************************************************************************
    * Program 	    : Master's Thesis - Soccer Table (Simulation)
    * Author  	    : Roman Parak
    * Created 	    : date ...
	* University    : Brno University of Technology(BUT)
	* Faculty       : Faculty of Mechanical Engineering(FME)
	* Study Program : Applied Computer Science and Control
	* Institute     : Institute of Automation and Computer Science
**********************************************************************************************
* Implementation OF PROGRAM simulation(rp_library/rp_funcx1/rp_functions.c)
**********************************************************************************************/

/************************************* LIBRARIES *********************************************/
#include <bur/plctypes.h>
#include <stdlib.h>
#include <stdio.h>
#include <math.h>

#ifdef __cplusplus
	extern "C"
	{
#endif
#include "rp_funcx1.h"
#ifdef __cplusplus
	};
#endif

/**********************************************************************************************************/
/************************************** FUNCTIONS & FUNCTIONS BLOCKS **************************************/
/**********************************************************************************************************/

signed short random_number(signed short min_num, signed short max_num)
{
    signed char result = 0,low_num = 0,high_num = 0;

    if(min_num < max_num){
        low_num  = min_num;
        high_num = max_num + 1;
    }else{
        low_num  = max_num + 1;
        high_num = min_num;
    }

    result = (rand()%(high_num - low_num)) + low_num;
    return result;

}// end function

void get_rotationalPostition(struct get_rotationalPostition* g_rP)
{
	LREAL mod_pos, lrealPart, x;
	int i;

	for(i = 0; i < (int)(sizeof(g_rP->actual_position)/sizeof(g_rP->actual_position[0])); i++){
		if((g_rP->actual_position[i] - g_rP->define_position[i]) == 0){
			g_rP->result[i] = 0;
		}else{
			if(fabs((g_rP->actual_position[i] - g_rP->define_position[i])) > 3600){
				x       = fabs((g_rP->actual_position[i] - g_rP->define_position[i]))/3600;
				mod_pos = modf(x,&lrealPart);

				if((g_rP->actual_position[i] - g_rP->define_position[i]) > 0){
					g_rP->result[i] = (g_rP->actual_position[i] - g_rP->define_position[i]) - (3600*lrealPart);
				}else{
					g_rP->result[i] = (g_rP->actual_position[i] - g_rP->define_position[i]) + (3600*lrealPart);
				}
			}else{
				g_rP->result[i] = fabs((g_rP->actual_position[i] - g_rP->define_position[i]));
			}
		}
	}

}// end function
```

#### Types.typ
```iecst
(*Enumerations*)

TYPE
	internal_turnPos : 	STRUCT
		auxiliary_move_pos : REAL;
		distance_ofMoveNeg : REAL;
		distance_ofMovePos : REAL;
		min_pos_ofAxes : ARRAY[0..3]OF REAL;
		max_pos_ofAxes : ARRAY[0..3]OF REAL;
		state : USINT;
	END_STRUCT;
	param_ac : 	STRUCT
		displacement : REAL;
		velocity : REAL;
		acceleration : REAL;
		deceleration : REAL;
	END_STRUCT;
	internal_ballShooting : 	STRUCT
		state : USINT;
	END_STRUCT;
	internal_controlAxis : 	STRUCT
		before_state : USINT;
		state : USINT;
	END_STRUCT;
	internal_startAxisR : 	STRUCT
		before_state : USINT;
		state : USINT;
	END_STRUCT;
	internal_machtInfo : 	STRUCT
		WINNER : USINT;
		DRAW : USINT;
		LOSE : USINT;
		length : UDINT;
		write_matchInfo : BOOL;
		auxiliary_str : ARRAY[0..10]OF UDINT;
		counter : USINT;
		results : ARRAY[0..1]OF DINT;
		UtcDTStructureGetTime_1 : UtcDTStructureGetTime;
		e_r_str : ARRAY[0..3]OF UDINT;
		DTStruct : DTStructure;
		state : USINT;
		before_state : USINT;
		string : ARRAY[0..8]OF STRING[25];
	END_STRUCT;
	match_info : 	STRUCT
		team_name_CPU : ARRAY[0..50]OF STRING[10];
		team_name_HUM : ARRAY[0..50]OF STRING[20];
		score_HUM : ARRAY[0..50]OF USINT;
		score_CPU : ARRAY[0..50]OF USINT;
		date : ARRAY[0..50]OF STRING[25];
	END_STRUCT;
	soccer_table_ENUM :
		(
		RST_EMPTY := -1,
		RST_INITIALIZATION_1 := 1,
		RST_INITIALIZATION_2 := 2,
		RST_INITIALIZATION_3 := 3,
		RST_INITIALIZATION_4 := 4,
		RST_INITIALIZATION_5 := 5,
		RST_INITIALIZATION_6 := 6,
		RST_INITIALIZATION_7 := 7,
		RST_INITIALIZATION_8 := 8,
		RST_INITIALIZATION_9 := 9,
		RST_INITIALIZATION_10 := 10,
		RST_INITIALIZATION_11 := 11,
		RST_INITIALIZATION_12 := 12,
		RST_CHECK_MODE := 13,
		RST_MANUAL_HOME := 14,
		RST_CALCULATION_DEFENSE := 15,
		RST_MOVE_INTO_DEFENSE_POS1 := 16,
		RST_MOVE_INTO_DEFENSE_POS2 := 17,
		RST_ATTACK_MODE_SHOOT1 := 20,
		RST_ATTACK_MODE_SHOOT2_GK := 21,
		RST_ATTACK_MODE_SHOOT3_GK := 22,
		RST_ATTACK_MODE_SHOOT2_DF := 23,
		RST_ATTACK_MODE_SHOOT3_DF := 24,
		RST_ATTACK_MODE_SHOOT2_MD := 25,
		RST_ATTACK_MODE_SHOOT3_MD := 26,
		RST_ATTACK_MODE_SHOOT2_FW := 27,
		RST_ATTACK_MODE_SHOOT3_FW := 28,
		RST_ATTACK_MODE_TURN_POS := 50,
		RST_RUN1 := 100,
		RST_RUN2 := 101,
		RST_RUN3 := 102,
		RST_RUN4 := 103,
		RST_RUN5 := 104,
		RST_SERVICE := 200,
		RST_STOP := 300,
		RST_AFTER_STOP := 301,
		RST_NULL_POS1 := 310,
		RST_NULL_POS2 := 311,
		RST_SAFETY := 400,
		RST_AFTER_SAFETY := 401,
		RST_AFTER_SAFETY_HOME := 402,
		RST_AFTER_SAFETY_N1 := 403,
		RST_AFTER_SAFETY_N2 := 404,
		RST_AFTER_SAFETY_N3 := 405,
		RST_AFTER_SAFETY_N4 := 406,
		RST_ERROR := 500,
		RST_ERROR2 := 501
		);
	rp_MainSteps :
		(
		STEP_INITIALIZATION0 := 0,
		STEP_INITIALIZATION1 := 1,
		STEP_INITIALIZATION2 := 2,
		STEP_INITIALIZATION3 := 3,
		STEP_INITIALIZATION4 := 4,
		STEP_INITIALIZATION5 := 5,
		STEP_INITIALIZATION6 := 6,
		STEP_INITIALIZATION7 := 7,
		STEP_INITIALIZATION8 := 8,
		STEP_START := 10,
		STEP_RUN1 := 100,
		STEP_RUN2 := 101,
		STEP_RUN3 := 102,
		STEP_RUN4 := 103,
		STEP_RUN5 := 104,
		STEP_RUN6 := 105,
		STEP_RUN7 := 106,
		STEP_RUN8 := 107,
		STEP_RUN9 := 108,
		STEP_RUN10 := 109,
		STEP_RUN11 := 110,
		STEP_RUN12 := 111,
		STEP_RUN13 := 112,
		STEP_RUN14 := 113,
		STEP_RUN15 := 114,
		STEP_RUN16 := 115,
		STEP_RUN17 := 116,
		STEP_RUN18 := 117,
		STEP_RUN19 := 118,
		STEP_RUN20 := 119,
		STEP_RUN21 := 120,
		STEP_RUN22 := 121,
		STEP_RUN23 := 122,
		STEP_RUN24 := 123,
		STEP_RUN25 := 124,
		STEP_RUN26 := 125,
		STEP_RUN27 := 126,
		STEP_RUN28 := 127,
		STEP_RUN29 := 128,
		STEP_RUN30 := 129,
		STEP_RUN31 := 130,
		STEP_RUN32 := 131,
		STEP_RUN33 := 132,
		STEP_RUN34 := 133,
		STEP_RUN35 := 134,
		STEP_RUN36 := 135,
		STEP_RUN37 := 136,
		STEP_RUN38 := 137,
		STEP_RUN39 := 138,
		STEP_RUN40 := 139,
		STEP_RUN41 := 140,
		STEP_RUN42 := 141,
		STEP_RUN43 := 142,
		STEP_RUN44 := 143,
		STEP_RUN45 := 144,
		STEP_RUN46 := 145,
		STEP_RUN47 := 146,
		STEP_RUN48 := 147,
		STEP_RUN49 := 148,
		STEP_RUN50 := 149,
		STEP_SERVICE1 := 200,
		STEP_SERVICE2 := 201,
		STEP_SERVICE3 := 202,
		STEP_STOP1 := 300,
		STEP_STOP2 := 301,
		STEP_STOP3 := 302,
		STEP_E_STOP := 350,
		STEP_ERROR1 := 400,
		STEP_ERROR2 := 401,
		STEP_ERROR3 := 402
		);
END_TYPE
```

#### forecast_direction.c
```c
/*********************************************************************************************
* B&R Automation - Perfection in Automation (https://www.br-automation.com)
    ******************************************************************************************
    * Program 	    : Master's Thesis - Soccer Table (Simulation)
    * Author  	    : Roman Parak
    * Created 	    : date ...
	* University    : Brno University of Technology(BUT)
	* Faculty       : Faculty of Mechanical Engineering(FME)
	* Study Program : Applied Computer Science and Control
	* Institute     : Institute of Automation and Computer Science
**********************************************************************************************
* Implementation OF PROGRAM simulation(rp_library/rp_funcx1/forecast_direction.c)
**********************************************************************************************/

/************************************* LIBRARIES *********************************************/
#include <bur/plctypes.h>
#include <math.h>

#ifdef __cplusplus
	extern "C"
	{
#endif
	#include "rp_funcx1.h"
#ifdef __cplusplus
	};
#endif

/**********************************************************************************************************/
/************************************** FUNCTIONS & FUNCTIONS BLOCKS **************************************/
/**********************************************************************************************************/

void forecast_direction(struct forecast_direction* f_d)
{
	USINT initial_state;
	UDINT auxiliary_str;

	struct calculate_directionOfTilt calc_dirOfTilt;
	struct calculate_nextDirection calc_nextDir;

	if((isnan(f_d->ball2_x)) && (isnan(f_d->ball2_y))){
		initial_state = 0;
	}else{
		initial_state = 1;
	}

	switch(initial_state){
		case 0:
			{
				f_d->first_reflectionX  = 0;
				f_d->first_reflectionY  = f_d->ball1_y;
				f_d->second_reflectionX = sqrt(-1);
				f_d->second_reflectionY = sqrt(-1);
				f_d->tilted       		= 0;

				auxiliary_str = (UDINT) strcpy(f_d->specific_direction,"straight");
			}
			break;
		case 1:
			{
				if(f_d->ball1_y == f_d->ball2_y){
					f_d->tilted = 0;

					if(f_d->ball1_x > f_d->ball2_x){
						auxiliary_str = (UDINT) strcpy(f_d->specific_direction,"straight-backward");

						f_d->first_reflectionX  = 0;
						f_d->first_reflectionY  = f_d->ball2_y;
						f_d->second_reflectionX = sqrt(-1);
						f_d->second_reflectionY = sqrt(-1);

					}else if(f_d->ball1_x < f_d->ball2_x){
						auxiliary_str = (UDINT) strcpy(f_d->specific_direction,"straight-forward");

						f_d->first_reflectionX  = 12100;
						f_d->first_reflectionY  = f_d->ball2_y;
						f_d->second_reflectionX = sqrt(-1);
						f_d->second_reflectionY = sqrt(-1);

					}else if(f_d->ball1_x == f_d->ball2_x){

						auxiliary_str = (UDINT) strcpy(f_d->specific_direction,"stopped");

						f_d->first_reflectionX  = f_d->ball1_x;
						f_d->first_reflectionY  = f_d->ball1_y;
						f_d->second_reflectionX = f_d->ball2_x;
						f_d->second_reflectionY = f_d->ball2_y;
					}
				}else{
					if(f_d->ball1_x == f_d->ball2_x){
						if(f_d->ball1_y < f_d->ball2_y){
							auxiliary_str = (UDINT) strcpy(f_d->specific_direction,"right");
						}else {
							auxiliary_str = (UDINT) strcpy(f_d->specific_direction,"left");
						}

						f_d->first_reflectionX  = f_d->ball1_x;
						f_d->first_reflectionY  = f_d->ball1_y;
						f_d->second_reflectionX = f_d->ball2_x;
						f_d->second_reflectionY = f_d->ball2_y;

					}else{
						f_d->tilted = 1;
						// input parameters into the function block calculate direction of tilt
						calc_dirOfTilt.ball1_x = f_d->ball1_x;
						calc_dirOfTilt.ball1_y = f_d->ball1_y;
						calc_dirOfTilt.ball2_x = f_d->ball2_x;
						calc_dirOfTilt.ball2_y = f_d->ball2_y;
						// call function block calculate direction of tilt
						calculate_directionOfTilt(&calc_dirOfTilt);
						// output parameters
						f_d->first_reflectionX  = calc_dirOfTilt.reflection_x;
						f_d->first_reflectionY  = calc_dirOfTilt.reflection_y;

						auxiliary_str = (UDINT) strcpy(f_d->specific_direction,calc_dirOfTilt.specific_direction);

						// input parameters into the function block calculate next direction
						calc_nextDir.ball2_x 			= f_d->ball2_x;
						calc_nextDir.ball2_y 			= f_d->ball2_y;
						calc_nextDir.first_reflection_x = calc_dirOfTilt.reflection_x;
						calc_nextDir.first_reflection_y = calc_dirOfTilt.reflection_y;
						calc_nextDir.state_ofDirection  = calc_dirOfTilt.state_ofDirection;
						// call function block calculate next direction
						calculate_nextDirection(&calc_nextDir);
						// output parameters
						f_d->second_reflectionX = calc_nextDir.second_reflection_x;
						f_d->second_reflectionY = calc_nextDir.second_reflection_y;
					}
				}
			}
			break;
	}// end switch

}// end function

void calculate_directionOfTilt(struct calculate_directionOfTilt* c_dT)
{
	USINT ball_direction;
	UDINT auxiliary_str;
	REAL distanceOfRatio_y, distanceOfRatio_x;
	REAL x_auxiliary, y_auxiliary;

	if((c_dT->ball2_y > c_dT->ball1_y) && (c_dT->ball2_x < c_dT->ball1_x)){
		ball_direction = 1;
		auxiliary_str = (UDINT) strcpy(c_dT->specific_direction,"up_backward");
	}else if((c_dT->ball2_y < c_dT->ball1_y) && (c_dT->ball2_x < c_dT->ball1_x)){
		ball_direction = 2;
		auxiliary_str = (UDINT) strcpy(c_dT->specific_direction,"down_backward");
	}else if((c_dT->ball2_y > c_dT->ball1_y) && (c_dT->ball2_x > c_dT->ball1_x)){
		ball_direction = 3;
		auxiliary_str = (UDINT) strcpy(c_dT->specific_direction,"up_forward");
	}else if((c_dT->ball2_y < c_dT->ball1_y) && (c_dT->ball2_x > c_dT->ball1_x)){
		ball_direction = 4;
		auxiliary_str = (UDINT) strcpy(c_dT->specific_direction,"down_forward");
	}

	switch(ball_direction){
		case 1:
			{
				// maximum of y : 3515
				// maximum of x : 0
				distanceOfRatio_y = ((3515 - c_dT->ball1_y)/(fabs(c_dT->ball1_y - c_dT->ball2_y)));
				distanceOfRatio_x = ((c_dT->ball1_x)/(fabs(c_dT->ball1_x - c_dT->ball2_x)));

				c_dT->state_ofDirection = ball_direction;

				x_auxiliary = c_dT->ball1_x - ((distanceOfRatio_y)*(fabs(c_dT->ball1_x - c_dT->ball2_x)));
				y_auxiliary = 3515;

				if((x_auxiliary >= 0) && (y_auxiliary <= 3515)){
					c_dT->reflection_x = x_auxiliary;
					c_dT->reflection_y = y_auxiliary;
				}else{
					c_dT->reflection_x = 0;
					c_dT->reflection_y = c_dT->ball1_y + ((distanceOfRatio_x)*(fabs(c_dT->ball1_y - c_dT->ball2_y)));
				}
			}
			break;
		case 2:
			{
				// maximum of y : -3515
				// maximum of x : 0
				distanceOfRatio_y = ((c_dT->ball1_y + 3515)/(fabs(c_dT->ball1_y - c_dT->ball2_y)));
				distanceOfRatio_x = ((c_dT->ball1_x)/(fabs(c_dT->ball1_x - c_dT->ball2_x)));

				c_dT->state_ofDirection = ball_direction;

				x_auxiliary = c_dT->ball1_x - ((distanceOfRatio_y)*(fabs(c_dT->ball1_x - c_dT->ball2_x)));
				y_auxiliary = -3515;

				if((x_auxiliary >= 0) && (y_auxiliary >= -3515)){
					c_dT->reflection_x = x_auxiliary;
					c_dT->reflection_y = y_auxiliary;
				}else{
					c_dT->reflection_x = 0;
					c_dT->reflection_y = c_dT->ball1_y - ((distanceOfRatio_x)*(fabs(c_dT->ball1_y - c_dT->ball2_y)));
				}
			}
			break;
		case 3:
			{
				// maximum of y : 3515
				// maximum of x : 12100
				distanceOfRatio_y = ((3515 - c_dT->ball1_y)/(fabs(c_dT->ball1_y - c_dT->ball2_y)));
				distanceOfRatio_x = ((12100 - c_dT->ball1_x)/(fabs(c_dT->ball1_x - c_dT->ball2_x)));

				c_dT->state_ofDirection = ball_direction;

				x_auxiliary = c_dT->ball1_x + ((distanceOfRatio_y)*(fabs(c_dT->ball1_x - c_dT->ball2_x)));
				y_auxiliary = 3515;

				if((x_auxiliary <= 12100) && (y_auxiliary <= 3515)){
					c_dT->reflection_x = x_auxiliary;
					c_dT->reflection_y = y_auxiliary;
				}else{
					c_dT->reflection_x = 12100;
					c_dT->reflection_y = c_dT->ball1_y + ((distanceOfRatio_x)*(fabs(c_dT->ball1_y-c_dT->ball2_y)));
				}
			}
			break;
		case 4:
			{
				// maximum of y : -3515
				// maximum of x : 12100
				distanceOfRatio_y = ((c_dT->ball1_y + 3515)/(fabs(c_dT->ball1_y - c_dT->ball2_y)));
				distanceOfRatio_x = ((12100 - c_dT->ball1_x)/(fabs(c_dT->ball1_x - c_dT->ball2_x)));

				c_dT->state_ofDirection = ball_direction;

				x_auxiliary = c_dT->ball1_x + ((distanceOfRatio_y)*(fabs(c_dT->ball1_x - c_dT->ball2_x)));
				y_auxiliary = -3515;

				if((x_auxiliary <= 12100) && (y_auxiliary >= -3515)){
					c_dT->reflection_x = x_auxiliary;
					c_dT->reflection_y = y_auxiliary;
				}else{
					c_dT->reflection_x = 12100;
					c_dT->reflection_y = c_dT->ball1_y - ((distanceOfRatio_x)*(fabs(c_dT->ball1_y - c_dT->ball2_y)));
				}
			}
			break;
	}// end switch

}// end function

void calculate_nextDirection(struct calculate_nextDirection* c_nD)
{
	REAL x_n, y_n;

	struct calculate_directionOfTilt calc_dT;

	switch(c_nD->state_ofDirection){
		case 1:
			{
				// direction : up, forward
				if(c_nD->first_reflection_x == 0){
					x_n = c_nD->first_reflection_x + (fabs(c_nD->first_reflection_x - c_nD->ball2_x)*(0.01));
					y_n = c_nD->first_reflection_y + (fabs(c_nD->first_reflection_y - c_nD->ball2_y)*(0.01));
				}else{
					x_n = c_nD->first_reflection_x - (fabs(c_nD->first_reflection_x - c_nD->ball2_x)*(0.01));
					y_n = c_nD->first_reflection_y - (fabs(c_nD->first_reflection_y - c_nD->ball2_y)*(0.01));
				}

				// input parameters into the function block calculate direction of tilt
				calc_dT.ball1_x = c_nD->first_reflection_x;
				calc_dT.ball1_y = c_nD->first_reflection_y;
				calc_dT.ball2_x = x_n;
				calc_dT.ball2_y = y_n;
				// call function block calculate direction of tilt
				calculate_directionOfTilt(&calc_dT);
				// output parameters
				c_nD->second_reflection_x = calc_dT.reflection_x;
				c_nD->second_reflection_y = calc_dT.reflection_y;
			}
			break;
		case 2:
			{
				// direction : down, forward
				if(c_nD->first_reflection_x == 0){
					x_n = c_nD->first_reflection_x + (fabs(c_nD->first_reflection_x - c_nD->ball2_x)*(0.01));
					y_n = c_nD->first_reflection_y - (fabs(c_nD->first_reflection_y - c_nD->ball2_y)*(0.01));
				}else{
					x_n = c_nD->first_reflection_x - (fabs(c_nD->first_reflection_x - c_nD->ball2_x)*(0.01));
					y_n = c_nD->first_reflection_y + (fabs(c_nD->first_reflection_y - c_nD->ball2_y)*(0.01));
				}

				// input parameters into the function block calculate direction of tilt
				calc_dT.ball1_x = c_nD->first_reflection_x;
				calc_dT.ball1_y = c_nD->first_reflection_y;
				calc_dT.ball2_x = x_n;
				calc_dT.ball2_y = y_n;
				// call function block calculate direction of tilt
				calculate_directionOfTilt(&calc_dT);
				// output parameters
				c_nD->second_reflection_x = calc_dT.reflection_x;
				c_nD->second_reflection_y = calc_dT.reflection_y;
			}
			break;
		case 3:
			{
				// direction : up, backward
				if(c_nD->first_reflection_x == 12100){
					x_n = c_nD->first_reflection_x - (fabs(c_nD->first_reflection_x - c_nD->ball2_x)*(0.01));
					y_n = c_nD->first_reflection_y + (fabs(c_nD->first_reflection_y - c_nD->ball2_y)*(0.01));
				}else{
					x_n = c_nD->first_reflection_x + (fabs(c_nD->first_reflection_x - c_nD->ball2_x)*(0.01));
					y_n = c_nD->first_reflection_y - (fabs(c_nD->first_reflection_y - c_nD->ball2_y)*(0.01));
				}

				// input parameters into the function block calculate direction of tilt
				calc_dT.ball1_x = c_nD->first_reflection_x;
				calc_dT.ball1_y = c_nD->first_reflection_y;
				calc_dT.ball2_x = x_n;
				calc_dT.ball2_y = y_n;
				// call function block calculate direction of tilt
				calculate_directionOfTilt(&calc_dT);
				// output parameters
				c_nD->second_reflection_x = calc_dT.reflection_x;
				c_nD->second_reflection_y = calc_dT.reflection_y;
			}
			break;
		case 4:
			{
				// direction : down, backward
				if(c_nD->first_reflection_x == 12100){
					x_n = c_nD->first_reflection_x - (fabs(c_nD->first_reflection_x - c_nD->ball2_x)*(0.01));
					y_n = c_nD->first_reflection_y - (fabs(c_nD->first_reflection_y - c_nD->ball2_y)*(0.01));
				}else{
					x_n = c_nD->first_reflection_x + (fabs(c_nD->first_reflection_x - c_nD->ball2_x)*(0.01));
					y_n = c_nD->first_reflection_y + (fabs(c_nD->first_reflection_y - c_nD->ball2_y)*(0.01));
				}

				// input parameters into the function block calculate direction of tilt
				calc_dT.ball1_x = c_nD->first_reflection_x;
				calc_dT.ball1_y = c_nD->first_reflection_y;
				calc_dT.ball2_x = x_n;
				calc_dT.ball2_y = y_n;
				// call function block calculate direction of tilt
				calculate_directionOfTilt(&calc_dT);
				// output parameters
				c_nD->second_reflection_x = calc_dT.reflection_x;
				c_nD->second_reflection_y = calc_dT.reflection_y;
			}
			break;
	}// end switch

}// end function
```

#### calculation_posDummies.c
```c
/*********************************************************************************************
* B&R Automation - Perfection in Automation (https://www.br-automation.com)
    ******************************************************************************************
    * Program 	    : Master's Thesis - Soccer Table (Simulation)
    * Author  	    : Roman Parak
    * Created 	    : date ...
	* University    : Brno University of Technology(BUT)
	* Faculty       : Faculty of Mechanical Engineering(FME)
	* Study Program : Applied Computer Science and Control
	* Institute     : Institute of Automation and Computer Science
**********************************************************************************************
* Implementation OF PROGRAM simulation(rp_library/rp_funcx1/calculation_posDummiesOpponent.c)
**********************************************************************************************/

/************************************* LIBRARIES *********************************************/
#include <bur/plctypes.h>
#ifdef __cplusplus
	extern "C"
	{
#endif
	#include "rp_funcx1.h"
#ifdef __cplusplus
	};
#endif

/**********************************************************************************************************/
/************************************** FUNCTIONS & FUNCTIONS BLOCKS **************************************/
/**********************************************************************************************************/

void calculation_posDummies(struct calculation_posDummies* c_pD)
{
	/*
		Args:
			INPUT
				displacemen : 	     displacement of individual axes()a
								     array of data type REAL, where the index of array is individual axis
								     e.g. goalkeeper has index 0 etc.
			OUTPUT
				gk_posD 		   : position dummy of the axis name Goalkeeper
									 1 position
				df_posD 		   : position dummies of the axis name Defender
									 2 positions
				md_posD 		   : position dummies of the axis name Midfielder
									 5 positions
				fw_posD 		   : position dummies of the axis name Forward
									 3 positions
				real_displacement  : real displacement, for example due to mistake at reading from the sensors
									 array of data type REAL - all output values
	*/

	/***************************************** declaration variables ****************************************/
	REAL max_dispOfD[4], min_dispOfD[4], matrix_posOfOpponent[4][5], actual_positions[4][5];
	USINT i,j;
	// Indexes : GK - 0, DF - 1, MD - 2, FW - 3
	// max displacement of dummies
	max_dispOfD[0] = c_pD->max_disp[0];
	max_dispOfD[1] = c_pD->max_disp[1];
	max_dispOfD[2] = c_pD->max_disp[2];
	max_dispOfD[3] = c_pD->max_disp[3];
	// min displacement of dummies
	min_dispOfD[0] = c_pD->min_disp[0];
	min_dispOfD[1] = c_pD->min_disp[1];
	min_dispOfD[2] = c_pD->min_disp[2];
	min_dispOfD[3] = c_pD->min_disp[3];
	// matrix of parameters
	// goalkeeper
	matrix_posOfOpponent[0][0] = 0;
	// defender
	matrix_posOfOpponent[1][0] = -1200;
	matrix_posOfOpponent[1][1] = 1200;
	// midfielder
	matrix_posOfOpponent[2][0] = -2400;
	matrix_posOfOpponent[2][1] = -1200;
	matrix_posOfOpponent[2][2] = 0;
	matrix_posOfOpponent[2][3] = 1200;
	matrix_posOfOpponent[2][4] = 2400;
	// forward
	matrix_posOfOpponent[3][0] = -2100;
	matrix_posOfOpponent[3][1] = 0;
	matrix_posOfOpponent[3][2] = 2100;

	/********************************************* calculation **********************************************/
	for(i = 0; i < (int)(sizeof(c_pD->displacement)/sizeof(c_pD->displacement[0])); i++){
		for(j = 0; j <= (int)(sizeof(c_pD->displacement)/sizeof(c_pD->displacement[0])); j++){
			if(c_pD->displacement[i] > max_dispOfD[i]){
				actual_positions[i][j] 	   = max_dispOfD[i] + matrix_posOfOpponent[i][j];
				c_pD->real_displacement[i] = max_dispOfD[i];
			}else if(c_pD->displacement[i] < min_dispOfD[i]){
				actual_positions[i][j] 	   = min_dispOfD[i] + matrix_posOfOpponent[i][j];
				c_pD->real_displacement[i] = min_dispOfD[i];
			}else{
				actual_positions[i][j]     = c_pD->displacement[i] + matrix_posOfOpponent[i][j];
				c_pD->real_displacement[i] = c_pD->displacement[i];
			}
		}
	}

	/**************************************** output real parameters ****************************************/
	// goalkeeper
	c_pD->actual_positionsOfDummies[0]  = actual_positions[0][0];
	// defender
	c_pD->actual_positionsOfDummies[1]  = actual_positions[1][0];
	c_pD->actual_positionsOfDummies[2]  = actual_positions[1][1];
	// midfielder
	c_pD->actual_positionsOfDummies[3]  = actual_positions[2][0];
	c_pD->actual_positionsOfDummies[4]  = actual_positions[2][1];
	c_pD->actual_positionsOfDummies[5]  = actual_positions[2][2];
	c_pD->actual_positionsOfDummies[6]  = actual_positions[2][3];
	c_pD->actual_positionsOfDummies[7]  = actual_positions[2][4];
	// forward
	c_pD->actual_positionsOfDummies[8]  = actual_positions[3][0];
	c_pD->actual_positionsOfDummies[9]  = actual_positions[3][1];
	c_pD->actual_positionsOfDummies[10] = actual_positions[3][2];

}// end function
```

#### calculation_crossingBall.c
```c
/*********************************************************************************************
* B&R Automation - Perfection in Automation (https://www.br-automation.com)
    ******************************************************************************************
    * Program 	    : Master's Thesis - Soccer Table (Simulation)
    * Author  	    : Roman Parak
    * Created 	    : date ...
	* University    : Brno University of Technology(BUT)
	* Faculty       : Faculty of Mechanical Engineering(FME)
	* Study Program : Applied Computer Science and Control
	* Institute     : Institute of Automation and Computer Science
**********************************************************************************************
* Implementation OF PROGRAM simulation(rp_library/rp_funcx1/calculation_crossingBall.c)
**********************************************************************************************/

/************************************* LIBRARIES *********************************************/
#include <bur/plctypes.h>
#include <stdio.h>
#include <stdlib.h>
#include <math.h>

#ifdef __cplusplus
	extern "C"
	{
#endif
	#include "rp_funcx1.h"
#ifdef __cplusplus
	};
#endif
// declaration function
int cmpfunc(const void *a, const void *b);

void calculation_crossingBall(struct calculation_crossingBall* c_cB)
{
	USINT initial_state;
	USINT count_aI[2];
	USINT i, s_i, t_iB1, t_iB1N, t_iB2, t_iB2N, i_aux, i_loaded, i_timeL, i_fbI, i_fbO;
	BOOL both_ball;
	REAL x_position[2], y_auxiliaryPos[4];
	REAL x_auxiliaryPos[4];

	struct arrival_timeOfBall a_tOfBall;

	x_auxiliaryPos[0] = c_cB->x_positions[0];
	x_auxiliaryPos[1] = c_cB->x_positions[1];
	x_auxiliaryPos[2] = c_cB->x_positions[2];
	x_auxiliaryPos[3] = c_cB->x_positions[3];

	c_cB->act_posOfAxesX[0] = x_auxiliaryPos[0];
	c_cB->act_posOfAxesX[1] = x_auxiliaryPos[1];
	c_cB->act_posOfAxesX[2] = x_auxiliaryPos[2];
	c_cB->act_posOfAxesX[3] = x_auxiliaryPos[3];

	x_position[0] = c_cB->ball1_x;
	x_position[1] = c_cB->first_reflection_x;

	if(isnan(c_cB->ball2_x) && isnan(c_cB->ball2_y)){
		both_ball = 0;
	}else{
		both_ball = 1;
	}

	for(i = 0; i < (int)(sizeof(x_position)/sizeof(x_position[0])); i++){
		if(x_position[i] > x_auxiliaryPos[3]){
			count_aI[i] = 4;
		}else if((x_position[i] > x_auxiliaryPos[2]) && (x_position[i] <= x_auxiliaryPos[3])){
			count_aI[i] = 3;
		}else if((x_position[i] > x_auxiliaryPos[1]) && (x_position[i] <= x_auxiliaryPos[2])){
			count_aI[i] = 2;
		}else if((x_position[i] > x_auxiliaryPos[0]) && (x_position[i] <= x_auxiliaryPos[1])){
			count_aI[i] = 1;
		}else{
			count_aI[i] = 0;
		}
	}

	c_cB->count_axesIntersection[0] = count_aI[0];
	c_cB->count_axesIntersection[1] = count_aI[1];

	if((fabs(c_cB->second_reflection_x - c_cB->first_reflection_x) < 1500) && (fabs(c_cB->first_reflection_x - c_cB->ball2_x) < 1500)){
		initial_state = 0;
	}else{
		if(c_cB->tilted == 1){
			initial_state = 1;
		}else{
			initial_state = 0;
		}
	}

	switch(initial_state){
		case 0:
			{
				// straight direction of ball
				for(s_i = 0; s_i < (int)(sizeof(y_auxiliaryPos)/sizeof(y_auxiliaryPos[0])); s_i++){
					if(both_ball == 1){
						c_cB->act_posOfAxesY[s_i] = c_cB->ball2_y;
					}else{
						c_cB->act_posOfAxesY[s_i] = c_cB->ball1_y;
					}
				}
			}
			break;
		case 1:
			{
				// tilted direction of ball
				if(c_cB->ball1_x > c_cB->ball2_x){
					for(t_iB1 = 0; t_iB1 < count_aI[0]; t_iB1++){
						if( t_iB1 < count_aI[1]){
							// down direction
							y_auxiliaryPos[t_iB1] = c_cB->first_reflection_y - (c_cB->first_reflection_y - c_cB->second_reflection_y)/((c_cB->first_reflection_x - c_cB->second_reflection_x)/(c_cB->first_reflection_x - x_auxiliaryPos[t_iB1]));
						}else{
							// up direction
							y_auxiliaryPos[t_iB1] = c_cB->ball2_y + ((c_cB->first_reflection_y - c_cB->ball2_y)/((c_cB->ball2_x - c_cB->first_reflection_x)/(c_cB->ball2_x - x_auxiliaryPos[t_iB1])));
						}
					}

					for(t_iB1N = count_aI[0]; t_iB1N < (int)(sizeof(y_auxiliaryPos)/sizeof(y_auxiliaryPos[0])); t_iB1N++){
						y_auxiliaryPos[t_iB1N] = c_cB->ball2_y;
					}
				}else{
					for(t_iB2 = count_aI[0]; t_iB2 < (int)(sizeof(y_auxiliaryPos)/sizeof(y_auxiliaryPos[0])); t_iB2++){
						if( t_iB2 < count_aI[1]){
							// up direction
							y_auxiliaryPos[t_iB2] = c_cB->ball2_y + (c_cB->first_reflection_y - c_cB->ball2_y)/((c_cB->ball2_x - c_cB->first_reflection_x)/(c_cB->ball2_x - x_auxiliaryPos[t_iB2]));
						}else{
							// down direction
							y_auxiliaryPos[t_iB2] = c_cB->first_reflection_y - (c_cB->first_reflection_y - c_cB->second_reflection_y)/((c_cB->first_reflection_x - c_cB->second_reflection_x)/(c_cB->first_reflection_x - x_auxiliaryPos[t_iB2]));
						}
					}

					for(t_iB2N = 0; t_iB2N < count_aI[0]; t_iB2N++){
						y_auxiliaryPos[t_iB2N] = c_cB->ball2_y;
					}
				}

				for(i_aux = 0; i_aux < (int)(sizeof(y_auxiliaryPos)/sizeof(y_auxiliaryPos[0])); i_aux++){
					if((y_auxiliaryPos[i_aux] < -3515) || (y_auxiliaryPos[i_aux] > 3515)){
						y_auxiliaryPos[i_aux] = c_cB->ball2_y;
					}
				}

				for(i_loaded = 0; i_loaded < (int)(sizeof(y_auxiliaryPos)/sizeof(y_auxiliaryPos[0])); i_loaded++){
					c_cB->act_posOfAxesY[i_loaded] = y_auxiliaryPos[i_loaded];
				}
			}
			break;

	}// end switch

	if((both_ball == 1 && count_aI[0] != 0) || (count_aI[1] != 0) || (x_auxiliaryPos[0] != 3800)){
		a_tOfBall.ball1_x 			 = c_cB->ball1_x;
		a_tOfBall.ball1_y 			 = c_cB->ball1_y;
		a_tOfBall.ball2_x 		     = c_cB->ball2_x;
		a_tOfBall.ball2_y 			 = c_cB->ball2_y;
		a_tOfBall.first_reflection_x = c_cB->first_reflection_x;
		a_tOfBall.first_reflection_y = c_cB->first_reflection_y;
		// input parameters into the function block arrival time of the ball
		for(i_fbI = 0; i_fbI < (int)(sizeof(y_auxiliaryPos)/sizeof(y_auxiliaryPos[0])); i_fbI++){
			a_tOfBall.act_posOfAxesX[i_fbI] = c_cB->act_posOfAxesX[i_fbI];
			a_tOfBall.act_posOfAxesY[i_fbI] = c_cB->act_posOfAxesY[i_fbI];
		}
	    a_tOfBall.time_B2B			 	      = c_cB->time_B2B;
		a_tOfBall.tilted	         		  = c_cB->tilted;
		a_tOfBall.count_axesIntersection[0]   = count_aI[0];
		a_tOfBall.count_axesIntersection[1]   = count_aI[1];
		// call function block arrival time of the ball
		arrival_timeOfBall(&a_tOfBall);
		// output parameters
		c_cB->overall_velocity = a_tOfBall.velocity;
		for(i_fbO = 0; i_fbO < (int)(sizeof(y_auxiliaryPos)/sizeof(y_auxiliaryPos[0])); i_fbO++){
			c_cB->time_axisIntersection[i_fbO] = a_tOfBall.time_aI[i_fbO];
		}

	}else{
		c_cB->overall_velocity = 150000;

		for(i_timeL = 0; i_timeL < (int)(sizeof(y_auxiliaryPos)/sizeof(y_auxiliaryPos[0])); i_timeL++){
			c_cB->time_axisIntersection[i_timeL] = fabs(x_auxiliaryPos[i_timeL] - x_position[0])/c_cB->overall_velocity ;
		}

	}
}// end function

void arrival_timeOfBall(struct arrival_timeOfBall* a_tOB)
{
	USINT initial_state;
	USINT i_eqS, i_B1S, i_B1Sn, i_OS, i_OSn, i_B1T, iB1Tn, iOT, iOTn;
	REAL time_f[4], previous_time;

	if(a_tOB->tilted == 1){
		initial_state = 1;
	}else{
		initial_state = 0;
	}

	switch(initial_state){
		case 0:
			{
				// straight direction of ball
				if(a_tOB->ball1_x == a_tOB->ball2_x){
					a_tOB->velocity = fabs((a_tOB->ball1_y - a_tOB->ball2_y))/a_tOB->time_B2B;

					for(i_eqS = 0; i_eqS < (int)(sizeof(a_tOB->act_posOfAxesX)/sizeof(a_tOB->act_posOfAxesX[0])); i_eqS++){
						a_tOB->time_aI[i_eqS] = fabs((a_tOB->ball1_y - a_tOB->ball2_y))/a_tOB->velocity;
					}

				}else if(a_tOB->ball1_x > a_tOB->ball2_x){
					a_tOB->velocity = fabs((a_tOB->ball1_x - a_tOB->ball2_x))/a_tOB->time_B2B;

					for(i_B1S = 0; i_B1S < a_tOB->count_axesIntersection[0]; i_B1S++){
						time_f[i_B1S] = fabs((a_tOB->ball2_x - a_tOB->act_posOfAxesX[i_B1S]))/a_tOB->velocity;
					}

					qsort(time_f,sizeof(time_f)/sizeof(time_f[0]),sizeof(REAL),cmpfunc);
					for(i_B1Sn = 0; i_B1Sn < (int)(sizeof(a_tOB->act_posOfAxesX)/sizeof(a_tOB->act_posOfAxesX[0])); i_B1Sn++){
						if(i_B1Sn < a_tOB->count_axesIntersection[0]){
							a_tOB->time_aI[i_B1Sn] = time_f[i_B1Sn];
						}else{
							a_tOB->time_aI[i_B1Sn] = a_tOB->time_B2B;
						}
					}
				}else{
					a_tOB->velocity = fabs((a_tOB->ball1_x - a_tOB->ball2_x))/a_tOB->time_B2B;

					if(a_tOB->ball2_x > 8300){
						for(i_OS = a_tOB->count_axesIntersection[0]; i_OS < (int)(sizeof(a_tOB->act_posOfAxesX)/sizeof(a_tOB->act_posOfAxesX[0])); i_OS++){
							a_tOB->time_aI[i_OS] = fabs((a_tOB->ball2_x - a_tOB->act_posOfAxesX[i_OS]))/a_tOB->velocity;
						}
					}else{
						for(i_OSn = 0; i_OSn < (int)(sizeof(a_tOB->act_posOfAxesX)/sizeof(a_tOB->act_posOfAxesX[0])); i_OSn++){
							a_tOB->time_aI[i_OSn] = a_tOB->time_B2B;
						}
					}
				}
			}
			break;
		case 1:
			{
				// tilted direction of ball
				a_tOB->velocity = sqrt(pow((a_tOB->ball1_x - a_tOB->ball2_x),2) + pow((a_tOB->ball1_y - a_tOB->ball2_y),2))/a_tOB->time_B2B;
				previous_time 	= sqrt(pow((a_tOB->ball2_x - a_tOB->first_reflection_x),2) + pow((a_tOB->ball2_y - a_tOB->first_reflection_y),2))/a_tOB->velocity;

				if(a_tOB->ball1_x > a_tOB->ball2_x){
					for(i_B1T = 0; i_B1T < a_tOB->count_axesIntersection[0]; i_B1T++){
						if(i_B1T < a_tOB->count_axesIntersection[1]){
							time_f[i_B1T] = sqrt(pow((a_tOB->first_reflection_x - a_tOB->act_posOfAxesX[i_B1T]),2) + pow((a_tOB->first_reflection_y - a_tOB->act_posOfAxesY[i_B1T]),2))/a_tOB->velocity + previous_time;
						}else{
							time_f[i_B1T] = sqrt(pow((a_tOB->ball2_x - a_tOB->act_posOfAxesX[i_B1T]),2) + pow((a_tOB->ball2_y - a_tOB->act_posOfAxesY[i_B1T]),2))/a_tOB->velocity;
						}
					}
					qsort(time_f,sizeof(time_f)/sizeof(time_f[0]),sizeof(REAL),cmpfunc);

					for(iB1Tn = 0; iB1Tn < (int)(sizeof(a_tOB->act_posOfAxesX)/sizeof(a_tOB->act_posOfAxesX[0])); iB1Tn++){
						if(iB1Tn < a_tOB->count_axesIntersection[0]){
							a_tOB->time_aI[iB1Tn] = time_f[iB1Tn];
						}else{
							a_tOB->time_aI[iB1Tn] = a_tOB->time_B2B;
						}
					}
				}else{
					for(iOT = a_tOB->count_axesIntersection[0]; iOT < (int)(sizeof(a_tOB->act_posOfAxesX)/sizeof(a_tOB->act_posOfAxesX[0])); iOT++){
						if(iOT < a_tOB->count_axesIntersection[1]){
							a_tOB->time_aI[iOT] = sqrt(pow((a_tOB->ball2_x - a_tOB->act_posOfAxesX[iOT]),2) + pow((a_tOB->ball2_y - a_tOB->act_posOfAxesY[iOT]),2))/a_tOB->velocity;
						}else{
							a_tOB->time_aI[iOT] = sqrt(pow((a_tOB->first_reflection_x - a_tOB->act_posOfAxesX[iOT]),2) + pow((a_tOB->first_reflection_y - a_tOB->act_posOfAxesY[iOT]),2))/a_tOB->velocity + previous_time;
						}
					}

					for(iOTn = 0; iOTn < a_tOB->count_axesIntersection[0]; iOTn++){
						a_tOB->time_aI[iOTn] = a_tOB->time_B2B;
					}
				}
			}
			break;
	}//end switch
}// end function

int cmpfunc(const void *a, const void *b)
{
	return (*(REAL*)b - *(REAL*)a);
}
```

#### calculation_displacementOfAxes.c
```c
/*********************************************************************************************
* B&R Automation - Perfection in Automation (https://www.br-automation.com)
    ******************************************************************************************
    * Program 	    : Master's Thesis - Soccer Table (Simulation)
    * Author  	    : Roman Parak
    * Created 	    : date ...
	* University    : Brno University of Technology(BUT)
	* Faculty       : Faculty of Mechanical Engineering(FME)
	* Study Program : Applied Computer Science and Control
	* Institute     : Institute of Automation and Computer Science
**********************************************************************************************
* Implementation OF PROGRAM simulation(rp_library/rp_funcx1/rp_functions.c)
**********************************************************************************************/

/************************************* LIBRARIES *********************************************/
#include <bur/plctypes.h>
#include <math.h>
#include <string.h>

#ifdef __cplusplus
	extern "C"
	{
#endif
	#include "rp_funcx1.h"
#ifdef __cplusplus
	};
#endif

void calculation_displacementOfAxes(struct calculation_displacementOfAxes* c_dOA)
{
	REAL max_dispOfD[4], min_dispOfD[4], max_posOfD[4], min_posOfD[4], matrix_posOfCPU[4][5], real_disp[4];
	REAL velocity[4], acceleration[4], deceleration[4];
	REAL aux_velocity[4], aux_acceleration[4];
	REAL aux_time;
	UDINT auxiliary_str;
	USINT i_rC, i_rCn, i, j, i_out, i_chRD, i_chRDn, i_chRDnn;

	struct calculation_realCrossing calc_rC;
	struct choosing_rightDummy ch_rightD;

	// Ceilings of the axes
	// Axes
	max_posOfD[0] = 820;
	max_posOfD[1] = 3050;
	max_posOfD[2] = 3050;
	max_posOfD[3] = 3055;

	min_posOfD[0] = -930;
	min_posOfD[1] = -3050;
	min_posOfD[2] = -3050;
	min_posOfD[3] = -3055;
	// Dummies {-50 units, without GK}
	max_dispOfD[0] = 800;
	max_dispOfD[1] = 1030;
	max_dispOfD[2] = 520;
	max_dispOfD[3] = 830;

	min_dispOfD[0] = -910;
	min_dispOfD[1] = -930;
	min_dispOfD[2] = -500;
	min_dispOfD[3] = -770;
	// Actual positions of dummies CPU
	// goalkeeper
	matrix_posOfCPU[0][0] = 0 + c_dOA->act_displacementCPU[0];
	// defender
	matrix_posOfCPU[1][0] = -1200 + c_dOA->act_displacementCPU[1];
	matrix_posOfCPU[1][1] = 1200 + c_dOA->act_displacementCPU[1];
	// midfielder
	matrix_posOfCPU[2][0] = -2400 + c_dOA->act_displacementCPU[2];
	matrix_posOfCPU[2][1] = -1200 + c_dOA->act_displacementCPU[2];
	matrix_posOfCPU[2][2] = 0 + c_dOA->act_displacementCPU[2];
	matrix_posOfCPU[2][3] = 1200 + c_dOA->act_displacementCPU[2];
	matrix_posOfCPU[2][4] = 2400 + c_dOA->act_displacementCPU[2];
	// forward
	matrix_posOfCPU[3][0] = -2100 + c_dOA->act_displacementCPU[3];
	matrix_posOfCPU[3][1] = 0 + c_dOA->act_displacementCPU[3];
	matrix_posOfCPU[3][2] = 2100 + c_dOA->act_displacementCPU[3];

	// function block -> output is a array of real crossing
	calc_rC.tilted = c_dOA->tilted;
	auxiliary_str = (UDINT) strcpy(calc_rC.specific_direction,c_dOA->specific_direction);
	for(i_rC = 0; i_rC < (int)(sizeof(max_posOfD)/sizeof(max_posOfD[0])); i_rC++){
		calc_rC.act_posOfAxesCPU_Y[i_rC]		 = c_dOA->act_posOfAxesCPU_Y[i_rC];
		calc_rC.act_posOfAxesHUM_Y[i_rC]		 = c_dOA->act_posOfAxesHUM_Y[i_rC];
		calc_rC.count_axesIntersectionHUM[i_rC]  = c_dOA->count_axesIntersectionHUM[i_rC];
		calc_rC.reversed_HUM[i_rC]				 = c_dOA->reversed_HUM[i_rC];
	}
	for(i_rCn = 0; i_rCn < (int)(sizeof(c_dOA->act_posOfDummiesH)/sizeof(c_dOA->act_posOfDummiesH[0])); i_rCn++){
		calc_rC.act_posOfDummiesH[i_rCn] = c_dOA->act_posOfDummiesH[i_rCn];
	}
	calc_rC.x_posOfBall[0] = c_dOA->x_posOfBall[0];
	calc_rC.x_posOfBall[1] = c_dOA->x_posOfBall[1];
	calculation_realCrossing(&calc_rC);

	for(i = 0; i < (int)(sizeof(calc_rC.real_cross)/sizeof(calc_rC.real_cross[0])); i++){
		if(calc_rC.real_cross[i] > max_dispOfD[i]){
			real_disp[i] = max_dispOfD[i];
		}else if(calc_rC.real_cross[i] < min_dispOfD[i] && calc_rC.real_cross[i] < max_dispOfD[i]){
			real_disp[i] = min_dispOfD[i];
		}else {
			ch_rightD.index      = i;
			ch_rightD.real_cross = calc_rC.real_cross[i];

			for(i_chRD = 0; i_chRD < (int)(sizeof(max_dispOfD)/sizeof(max_dispOfD[0])); i_chRD++){
				ch_rightD.max_dispOfD[i_chRD] = max_dispOfD[i_chRD];
				ch_rightD.min_dispOfD[i_chRD] = min_dispOfD[i_chRD];
			}

			for(i_chRDn = 0; i_chRDn < (int)(sizeof(max_dispOfD)/sizeof(max_dispOfD[0])); i_chRDn++){
				for(i_chRDnn = 0; i_chRDnn <= (int)(sizeof(max_dispOfD)/sizeof(max_dispOfD[0]));i_chRDnn++){
					ch_rightD.matrix_posOfCPU[i_chRDn][i_chRDnn] = matrix_posOfCPU[i_chRDn][i_chRDnn];
				}
			}
			choosing_rightDummy(&ch_rightD);

			real_disp[i] = ch_rightD.actual_displacement;
		}
	}// end for{i}

	for(i_out = 0; i_out < (int)(sizeof(calc_rC.real_cross)/sizeof(calc_rC.real_cross[0])); i_out++){
		// max velocity = 29000, max acceleration = 489 000
		aux_time = 0.07;
		aux_velocity[i_out] = fabs(fabs(real_disp[i_out]) - fabs(c_dOA->act_displacementCPU[i_out]))/c_dOA->time_axisIntersection[i_out];

		if(aux_velocity[i_out] > 29000){
			velocity[i_out] 		= fabs(fabs(real_disp[i_out]) - fabs(c_dOA->act_displacementCPU[i_out]))/aux_time;
			aux_acceleration[i_out] = velocity[i_out]/c_dOA->time_axisIntersection[i_out];

			if(aux_acceleration[i_out] > 489000){
				acceleration[i_out] = 489000;
				deceleration[i_out] = 489000;
			}else{
				acceleration[i_out] = aux_acceleration[i_out];
				deceleration[i_out] = aux_acceleration[i_out];
			}
		}else{
			velocity[i_out] 		= aux_velocity[i_out];
			aux_acceleration[i_out] = velocity[i_out]/c_dOA->time_axisIntersection[i_out];

			if(aux_acceleration[i_out] > 489000){
				acceleration[i_out] = 489000;
				deceleration[i_out] = 489000;
			}else{
				acceleration[i_out] = aux_acceleration[i_out];
				deceleration[i_out] = aux_acceleration[i_out];
			}
		}

		if(real_disp[i_out] > max_dispOfD[i_out]){
			c_dOA->displacement[i_out] = max_dispOfD[i_out];
		}else if(real_disp[i_out] < min_dispOfD[i_out] && real_disp[i_out] < max_dispOfD[i_out]){
			c_dOA->displacement[i_out] = min_dispOfD[i_out];
		}else{
			c_dOA->displacement[i_out] = real_disp[i_out];
		}
		c_dOA->velocity[i_out] 	   = velocity[i_out];
		c_dOA->acceleration[i_out] = acceleration[i_out];
		c_dOA->deceleration[i_out] = deceleration[i_out];
	}// end for{i_out}

}// end function

void calculation_realCrossing(struct calculation_realCrossing* c_rC)
{
	REAL matrix_posOfHUM[4][5], matrix_crossH_Iter[0][5], matrix_crossH_Pos[0][5];
	REAL predicted_pos;
	USINT number_ofD[4], count_crossH, count_calcH;
	USINT iteration, iteration_positionH;
	USINT j, j_null, i_yC, i_yCn, i_cNC, i_out, r;
	BOOL auxiliary_bool,auxiliary_boolNo2;
	UDINT auxiliary_str;

	struct calculation_newCrossing calc_newC;

	auxiliary_bool 	  = 0;
	auxiliary_boolNo2 = 0;
	// Actual positions of dummies HUMAN
	// goalkeeper
	matrix_posOfHUM[0][0] = c_rC->act_posOfDummiesH[0];
	// defender
	matrix_posOfHUM[1][0] = c_rC->act_posOfDummiesH[1];
	matrix_posOfHUM[1][1] = c_rC->act_posOfDummiesH[2];
	// midfielder
	matrix_posOfHUM[2][0] = c_rC->act_posOfDummiesH[3];
	matrix_posOfHUM[2][1] = c_rC->act_posOfDummiesH[4];
	matrix_posOfHUM[2][2] = c_rC->act_posOfDummiesH[5];
	matrix_posOfHUM[2][3] = c_rC->act_posOfDummiesH[6];
	matrix_posOfHUM[2][4] = c_rC->act_posOfDummiesH[7];
	// forward
	matrix_posOfHUM[3][0] = c_rC->act_posOfDummiesH[8];
	matrix_posOfHUM[3][1] = c_rC->act_posOfDummiesH[9];
	matrix_posOfHUM[3][2] = c_rC->act_posOfDummiesH[10];

	number_ofD[0] = 1;
	number_ofD[1] = 2;
	number_ofD[2] = 5;
	number_ofD[3] = 3;

	calc_newC.reversed_HUM = 1;

	count_crossH   = c_rC->count_axesIntersectionHUM[0];
	count_calcH    = 5 - count_crossH;

	if(count_calcH == 0){
		iteration = 1;
	}else{
		iteration = count_calcH;
	}

	if(count_calcH < 5){
		for(j = 0; j < number_ofD[count_calcH - 1]; j++){
			if(c_rC->reversed_HUM[count_calcH - 1] == 0){
				if(((matrix_posOfHUM[count_calcH - 1][j] <= c_rC->act_posOfAxesHUM_Y[count_calcH - 1] + 100) && (matrix_posOfHUM[count_calcH - 1][j] >= c_rC->act_posOfAxesHUM_Y[count_calcH - 1])) && (matrix_posOfHUM[count_calcH - 1][j] != c_rC->act_posOfAxesHUM_Y[count_calcH - 1])){
					matrix_crossH_Iter[0][j] = count_calcH;
					matrix_crossH_Pos[0][j]  = fabs(fabs(matrix_posOfHUM[count_calcH - 1][j]) - fabs(c_rC->act_posOfAxesHUM_Y[count_calcH - 1]));
				}else if(((matrix_posOfHUM[count_calcH - 1][j] >= c_rC->act_posOfAxesHUM_Y[count_calcH - 1] - 100) && (matrix_posOfHUM[count_calcH - 1][j] <= c_rC->act_posOfAxesHUM_Y[count_calcH - 1])) && (matrix_posOfHUM[count_calcH - 1][j] != c_rC->act_posOfAxesHUM_Y[count_calcH - 1])){
					matrix_crossH_Iter[0][j] = count_calcH;
					matrix_crossH_Pos[0][j]  = (-1)*fabs(fabs(matrix_posOfHUM[count_calcH - 1][j]) - fabs(c_rC->act_posOfAxesHUM_Y[count_calcH - 1]));
				}else if(matrix_posOfHUM[count_calcH - 1][j] == c_rC->act_posOfAxesHUM_Y[count_calcH - 1]){
					matrix_crossH_Iter[0][j] = count_calcH;
					matrix_crossH_Pos[0][j]  = 0;
				}else{
					matrix_crossH_Iter[0][j] = 0;
					matrix_crossH_Pos[0][j]  = 0;
				}
			}else{
				matrix_crossH_Iter[0][j] = 0;
				matrix_crossH_Pos[0][j]  = 0;
			}
		}

		for(r = 0; r < number_ofD[count_calcH - 1]; r++){
			if(matrix_crossH_Iter[0][r] != 0){
				calc_newC.reversed_HUM = 0;
			}
		}
		for(j_null = 0; j_null < number_ofD[count_calcH - 1]; j_null++){
			if(matrix_crossH_Iter[0][j_null] != 0){
				auxiliary_bool 		= 1;
				predicted_pos  		= matrix_crossH_Pos[0][j_null];
				iteration_positionH = matrix_crossH_Iter[0][j_null];
			}
		}

		if(auxiliary_bool == 0){
			if(c_rC->tilted == 0){
				predicted_pos 		= 0;
				iteration_positionH = iteration;
			}else{
				auxiliary_boolNo2 = 1;
				for(i_yCn = 0; i_yCn < (int)(sizeof(c_rC->act_posOfAxesCPU_Y)/sizeof(c_rC->act_posOfAxesCPU_Y[0])); i_yCn++){
					c_rC->real_cross[i_yCn] = c_rC->act_posOfAxesCPU_Y[i_yCn];
				}
			}
		}

	}else{
		if(c_rC->tilted == 0){
			calc_newC.reversed_HUM = 0;
			predicted_pos 		   = 0;
			iteration_positionH    = count_calcH;
		}else{
			auxiliary_boolNo2 = 1;
			for(i_yC = 0; i_yC < (int)(sizeof(c_rC->act_posOfAxesCPU_Y)/sizeof(c_rC->act_posOfAxesCPU_Y[0])); i_yC++){
				c_rC->real_cross[i_yC] = c_rC->act_posOfAxesCPU_Y[i_yC];
			}
		}
	}// end : if(count_calcH < 5)

	if(auxiliary_boolNo2 != 1){
		auxiliary_str = (UDINT) strcpy(calc_newC.specific_direction,c_rC->specific_direction);
		calc_newC.iteration 		 = iteration_positionH;
		calc_newC.predicted_position = predicted_pos;
		for(i_cNC = 0; i_cNC < (int)(sizeof(c_rC->act_posOfAxesCPU_Y)/sizeof(c_rC->act_posOfAxesCPU_Y[0])); i_cNC++){
			calc_newC.act_posOfAxesCPU_Y[i_cNC] = c_rC->act_posOfAxesCPU_Y[i_cNC];
			calc_newC.act_posOfAxesHUM_Y[i_cNC] = c_rC->act_posOfAxesHUM_Y[i_cNC];
		}
		calc_newC.x_posOfBall[0] = c_rC->x_posOfBall[0];
		calc_newC.x_posOfBall[1] = c_rC->x_posOfBall[1];
		calculation_newCrossing(&calc_newC);

		for(i_out = 0; i_out < (int)(sizeof(c_rC->act_posOfAxesCPU_Y)/sizeof(c_rC->act_posOfAxesCPU_Y[0])); i_out++){
			c_rC->real_cross[i_out] = calc_newC.new_cross[i_out];
		}
	}// end if(auxiliary_boolNo2 != 1)
}// end function

void calculation_newCrossing(struct calculation_newCrossing* c_nC)
{
	INT gk_max, gk_min, value;
	SINT iteration;
	DINT resultUP, resultLF, resultDOWN, resultRH;
	REAL y_crossGK, y_crossDF, y_crossMD, y_crossFW;

	// initial max goalkeeper
	gk_max = 800;
	gk_min = -910;

	resultUP   = strcmp(c_nC->specific_direction, "up_backward");
	resultLF   = strcmp(c_nC->specific_direction, "left");
	resultDOWN = strcmp(c_nC->specific_direction, "down_backward");
	resultRH   = strcmp(c_nC->specific_direction, "right");

	if(resultUP == 0 || resultLF == 0){
		value = 200;
	}else if(resultDOWN == 0 || resultRH == 0){
		value = -200;
	}else{
		value = 200;
	}

	if(c_nC->iteration > 4){
		iteration = 4;
	}else{
		iteration = c_nC->iteration;
	}

	switch(iteration){
		case 1:
			{
				y_crossFW = c_nC->act_posOfAxesCPU_Y[4];
				y_crossMD = y_crossFW + value;
				y_crossDF = y_crossMD + value;
				y_crossGK = y_crossDF + value;

				if(fabs(y_crossGK) > fabs(y_crossFW)){
					y_crossGK = y_crossFW - value;
				}

				if(fabs(y_crossMD) < fabs(y_crossFW)){
					y_crossMD = y_crossFW - value;
					y_crossDF = y_crossMD - value;
				}
			}
			break;
		case 2:
			{
				if(c_nC->x_posOfBall[0] >= 9800){
					y_crossFW = c_nC->act_posOfAxesHUM_Y[iteration] - c_nC->predicted_position;
					y_crossMD = y_crossFW + value;
					y_crossDF = y_crossMD + value;
					y_crossGK = y_crossDF + value;

					if(fabs(y_crossGK) > fabs(y_crossFW)){
						y_crossGK = y_crossFW - value;
					}

					if(fabs(y_crossMD) < fabs(y_crossFW)){
						y_crossMD = y_crossFW - value;
						y_crossDF = y_crossMD - value;
					}
				}else{
					y_crossFW = c_nC->act_posOfAxesHUM_Y[3] - c_nC->predicted_position;
					y_crossMD = y_crossFW + value;
					y_crossDF = y_crossMD + value;
					y_crossGK = y_crossDF + value;

					if(fabs(y_crossGK) > fabs(y_crossFW)){
						y_crossGK = y_crossFW - value;
					}

					if(fabs(y_crossMD) < fabs(y_crossFW)){
						y_crossMD = y_crossFW - value;
						y_crossDF = y_crossMD - value;
					}
				}
			}
			break;
		case 3:
			{
				if(c_nC->reversed_HUM == 1){
					y_crossFW = c_nC->act_posOfAxesHUM_Y[3] - c_nC->predicted_position;
					y_crossMD = y_crossFW + value;
				}else{
					y_crossFW = c_nC->act_posOfAxesHUM_Y[3] - c_nC->predicted_position;
					y_crossMD = y_crossFW + value;
				}

				y_crossDF = y_crossMD + value;
				y_crossGK = y_crossFW + value;

				if(fabs(y_crossGK) > fabs(y_crossFW)){
					y_crossGK = y_crossFW - value;
				}

				if(fabs(y_crossMD) < fabs(y_crossFW)){
					y_crossMD = y_crossFW - value;
					y_crossDF = y_crossMD - value;
				}
			}
			break;
		case 4:
			{
				if(c_nC->x_posOfBall[0] >= 5300){
					if(c_nC->reversed_HUM == 1){
						y_crossFW = c_nC->act_posOfAxesCPU_Y[3] - c_nC->predicted_position;
						y_crossMD = c_nC->act_posOfAxesCPU_Y[2] - c_nC->predicted_position;
						y_crossDF = y_crossMD + value;
						y_crossGK = y_crossFW + value;
					}else{
						y_crossFW = c_nC->act_posOfAxesCPU_Y[3] - c_nC->predicted_position;
						y_crossMD = c_nC->act_posOfAxesCPU_Y[2] - c_nC->predicted_position;
						y_crossDF = y_crossMD - c_nC->predicted_position;
						y_crossGK = y_crossFW + value;

					}

					if(fabs(y_crossGK) > fabs(y_crossFW)){
						y_crossGK = y_crossFW - value;
					}
					if(fabs(y_crossMD) < fabs(y_crossFW)){
						y_crossDF = y_crossMD - value;
					}
				}else{
					y_crossFW = c_nC->act_posOfAxesCPU_Y[3] - c_nC->predicted_position;
					y_crossMD = c_nC->act_posOfAxesCPU_Y[2] - c_nC->predicted_position;
					y_crossDF = y_crossMD - c_nC->predicted_position;
					y_crossGK = y_crossFW + value;
				}

				if(c_nC->x_posOfBall[0] <= 2300){
					y_crossGK = c_nC->act_posOfAxesCPU_Y[0];
				}
			}
			break;
	}// end switch

	if(y_crossGK > gk_max){
		y_crossGK = y_crossDF - 200;
	}else if(y_crossGK < gk_min){
		y_crossGK = y_crossDF + 200;
	}

	//c_nC->new_cross[0] = y_crossGK;

	if(c_nC->act_posOfAxesCPU_Y[0] > gk_max){
		c_nC->new_cross[0] = gk_max;
	}else if(c_nC->act_posOfAxesCPU_Y[0] < gk_min){
		c_nC->new_cross[0] = gk_min;
	}else{
		c_nC->new_cross[0] = c_nC->act_posOfAxesCPU_Y[0];
	}

	c_nC->new_cross[1] = y_crossDF;
	c_nC->new_cross[2] = y_crossMD;
	c_nC->new_cross[3] = y_crossFW;

}// end function

void choosing_rightDummy(struct choosing_rightDummy* ch_rD)
{
	REAL real_cross;
	REAL d_DFD[2],d_MDD[5], d_FWD[3];
	USINT i_df, i_md, i_fw;
	struct calculete_min calc_m;

	switch(ch_rD->index){
		case 0:
			{
				real_cross 				   = ch_rD->real_cross;
				ch_rD->actual_displacement = real_cross;
			}
			break;
		case 1:
			{
				d_DFD[0] = fabs((fabs(ch_rD->matrix_posOfCPU[ch_rD->index][0]) + ch_rD->real_cross));
				d_DFD[1] = fabs((ch_rD->matrix_posOfCPU[ch_rD->index][1] - ch_rD->real_cross));

				for(i_df = 0; i_df < (int)(sizeof(calc_m.cmp_num)/sizeof(calc_m.cmp_num[0])); i_df++){
					if(i_df < ((int)(sizeof(d_DFD)/sizeof(d_DFD[0])))){
						calc_m.cmp_num[i_df] = d_DFD[i_df];
					}else{
						calc_m.cmp_num[i_df] = 5000;
					}
				}
			}
			break;
		case 2:
			{
				d_MDD[0] = fabs((fabs(ch_rD->matrix_posOfCPU[ch_rD->index][0]) + ch_rD->real_cross));
				d_MDD[1] = fabs((fabs(ch_rD->matrix_posOfCPU[ch_rD->index][1]) + ch_rD->real_cross));
				d_MDD[2] = fabs((ch_rD->real_cross));
				d_MDD[3] = fabs((fabs(ch_rD->matrix_posOfCPU[ch_rD->index][3]) - ch_rD->real_cross));
				d_MDD[4] = fabs((fabs(ch_rD->matrix_posOfCPU[ch_rD->index][4]) - ch_rD->real_cross));

				for(i_md = 0; i_md < (int)(sizeof(calc_m.cmp_num)/sizeof(calc_m.cmp_num[0])); i_md++){
					calc_m.cmp_num[i_md] = d_MDD[i_md];
				}
			}
			break;
		case 3:
			{
				d_FWD[0] = fabs((fabs(ch_rD->matrix_posOfCPU[ch_rD->index][0]) + ch_rD->real_cross));
				d_FWD[1] = fabs((ch_rD->real_cross));
				d_FWD[2] = fabs((fabs(ch_rD->matrix_posOfCPU[ch_rD->index][2]) - ch_rD->real_cross));

				for(i_fw = 0; i_fw < (int)(sizeof(calc_m.cmp_num)/sizeof(calc_m.cmp_num[0])); i_fw++){
					if(i_fw < ((int)(sizeof(d_FWD)/sizeof(d_FWD[0])))){
						calc_m.cmp_num[i_fw] = d_FWD[i_fw];
					}else{
						calc_m.cmp_num[i_fw] = 5000;
					}
				}
			}
			break;
	}// end switch

	if(ch_rD->index != 0){
		calculete_min(&calc_m);

		if(calc_m.number > ch_rD->max_dispOfD[ch_rD->index]){
			real_cross = ch_rD->max_dispOfD[ch_rD->index];
		}else if(calc_m.number < ch_rD->min_dispOfD[ch_rD->index]){
			real_cross = ch_rD->min_dispOfD[ch_rD->index];
		}else{
			real_cross = calc_m.number;
		}

		if(ch_rD->real_cross > ch_rD->matrix_posOfCPU[ch_rD->index][calc_m.index]){
			ch_rD->actual_displacement = real_cross;
		}else{
			ch_rD->actual_displacement = (-1)*real_cross;
		}
	}
}// end function

void calculete_min(struct calculete_min* c_m)
{
	REAL min;
	USINT i, idx;

	min = 30000;
	for(i = 0; i < (int)(sizeof(c_m->cmp_num)/sizeof(c_m->cmp_num[0])); i++){
		if(c_m->cmp_num[i] < min){
			min = c_m->cmp_num[i];
			idx = i;
		}
	}

	c_m->index  = idx;
	c_m->number = min;
}// end function
```
